gfCNCPoint1[15648] = {X 518.0643, Y 36.2972, Z -1.3333, A 0.000, B 0.000, C 0.000 }
gfCNCPoint1[15649] = {X 518.9098, Y 36.0014, Z -1.3333, A 0.000, B 0.000, C 0.000 }
gfCNCPoint1[15650] = {X 519.7999, Y 35.9011, Z -1.3333, A 0.000, B 0.000, C 0.000 }
gfCNCPoint1[15651] = {X 520.5225, Y 35.9015, Z -1.3333, A 0.000, B 0.000, C 0.000 }
gfCNCPoint1[15652] = {X 521.3209, Y 35.9930, Z -1.3333, A 0.000, B 0.000, C 0.000 }
gfCNCPoint1[15653] = {X 522.0848, Y 36.2423, Z -1.3333, A 0.000, B 0.000, C 0.000 }
gfCNCPoint1[15654] = {X 522.7835, Y 36.6393, Z -1.3333, A 0.000, B 0.000, C 0.000 }
gfCNCPoint1[15655] = {X 523.3887, Y 37.1679, Z -1.3333, A 0.000, B 0.000, C 0.000 }
gfCNCPoint1[15656] = {X 523.8761, Y 37.8068, Z -1.3333, A 0.000, B 0.000, C 0.000 }
gfCNCPoint1[15657] = {X 534.9519, Y 37.8074, Z -1.3333, A 0.000, B 0.000, C 0.000 }
gfCNCPoint1[15658] = {X 534.9519, Y 34.0445, Z -1.3333, A 0.000, B 0.000, C 0.000 }
gfCNCPoint1[15659] = {X 534.9533, Y 33.6446, Z -1.3333, A 0.000, B 0.000, C 0.000 }
gfCNCPoint1[15660] = {X 529.9327, Y 33.6439, Z -1.3333, A 0.000, B 0.000, C 0.000 }
gfCNCPoint1[15661] = {X 529.8235, Y 33.8172, Z -1.3333, A 0.000, B 0.000, C 0.000 }
gfCNCPoint1[15662] = {X 529.1840, Y 34.5408, Z -1.3333, A 0.000, B 0.000, C 0.000 }
gfCNCPoint1[15663] = {X 528.3897, Y 35.0900, Z -1.3333, A 0.000, B 0.000, C 0.000 }
gfCNCPoint1[15664] = {X 527.4869, Y 35.4329, Z -1.3333, A 0.000, B 0.000, C 0.000 }
gfCNCPoint1[15665] = {X 526.5282, Y 35.5495, Z -1.3333, A 0.000, B 0.000, C 0.000 }
gfCNCPoint1[15666] = {X 525.8868, Y 35.5495, Z -1.3333, A 0.000, B 0.000, C 0.000 }
gfCNCPoint1[15667] = {X 524.9967, Y 35.4492, Z -1.3333, A 0.000, B 0.000, C 0.000 }
gfCNCPoint1[15668] = {X 524.1512, Y 35.1533, Z -1.3333, A 0.000, B 0.000, C 0.000 }
gfCNCPoint1[15669] = {X 523.3928, Y 34.6768, Z -1.3333, A 0.000, B 0.000, C 0.000 }
gfCNCPoint1[15670] = {X 522.7594, Y 34.0434, Z -1.3333, A 0.000, B 0.000, C 0.000 }
gfCNCPoint1[15671] = {X 522.2829, Y 33.2850, Z -1.3333, A 0.000, B 0.000, C 0.000 }
gfCNCPoint1[15672] = {X 521.9870, Y 32.4395, Z -1.3333, A 0.000, B 0.000, C 0.000 }
gfCNCPoint1[15673] = {X 521.8868, Y 31.5495, Z -1.3333, A 0.000, B 0.000, C 0.000 }
gfCNCPoint1[15674] = {X 521.8868, Y 24.5714, Z -1.3333, A 0.000, B 0.000, C 0.000 }
gfCNCPoint1[15675] = {X 521.9870, Y 23.6813, Z -1.3333, A 0.000, B 0.000, C 0.000 }
gfCNCPoint1[15676] = {X 522.2829, Y 22.8359, Z -1.3333, A 0.000, B 0.000, C 0.000 }
gfCNCPoint1[15677] = {X 522.7594, Y 22.0775, Z -1.3333, A 0.000, B 0.000, C 0.000 }
gfCNCPoint1[15678] = {X 523.3928, Y 21.4441, Z -1.3333, A 0.000, B 0.000, C 0.000 }
gfCNCPoint1[15679] = {X 524.1512, Y 20.9675, Z -1.3333, A 0.000, B 0.000, C 0.000 }
gfCNCPoint1[15680] = {X 524.9967, Y 20.6717, Z -1.3333, A 0.000, B 0.000, C 0.000 }
gfCNCPoint1[15681] = {X 525.8868, Y 20.5714, Z -1.3333, A 0.000, B 0.000, C 0.000 }
gfCNCPoint1[15682] = {X 526.5664, Y 20.5716, Z -1.3333, A 0.000, B 0.000, C 0.000 }
gfCNCPoint1[15683] = {X 527.3632, Y 20.6595, Z -1.3333, A 0.000, B 0.000, C 0.000 }
gfCNCPoint1[15684] = {X 528.1265, Y 20.9045, Z -1.3333, A 0.000, B 0.000, C 0.000 }
gfCNCPoint1[15685] = {X 528.8256, Y 21.2968, Z -1.3333, A 0.000, B 0.000, C 0.000 }
gfCNCPoint1[15686] = {X 529.4324, Y 21.8207, Z -1.3333, A 0.000, B 0.000, C 0.000 }
gfCNCPoint1[15687] = {X 529.9226, Y 22.4550, Z -1.3333, A 0.000, B 0.000, C 0.000 }
gfCNCPoint1[15688] = {X 534.9519, Y 22.4554, Z -1.3333, A 0.000, B 0.000, C 0.000 }
gfCNCPoint1[15689] = {X 534.9519, Y 19.7809, Z -1.3333, A 0.000, B 0.000, C 0.000 }
gfCNCPoint1[15690] = {X 534.9534, Y 19.3810, Z -1.3333, A 0.000, B 0.000, C 0.000 }
gfCNCPoint1[15691] = {X 524.0161, Y 19.3804, Z -1.3333, A 0.000, B 0.000, C 0.000 }
gfCNCPoint1[15692] = {X 523.9057, Y 19.5536, Z -1.3333, A 0.000, B 0.000, C 0.000 }
gfCNCPoint1[15693] = {X 523.2662, Y 20.2771, Z -1.3333, A 0.000, B 0.000, C 0.000 }
gfCNCPoint1[15694] = {X 522.4720, Y 20.8263, Z -1.3333, A 0.000, B 0.000, C 0.000 }
gfCNCPoint1[15695] = {X 521.5693, Y 21.1692, Z -1.3333, A 0.000, B 0.000, C 0.000 }
gfCNCPoint1[15696] = {X 520.6107, Y 21.2857, Z -1.3333, A 0.000, B 0.000, C 0.000 }
gfCNCPoint1[15697] = {X 519.9691, Y 21.2857, Z -1.3333, A 0.000, B 0.000, C 0.000 }
gfCNCPoint1[15698] = {X 519.0790, Y 21.1854, Z -1.3333, A 0.000, B 0.000, C 0.000 }
gfCNCPoint1[15699] = {X 518.2336, Y 20.8896, Z -1.3333, A 0.000, B 0.000, C 0.000 }
gfCNCPoint1[15700] = {X 517.4751, Y 20.4130, Z -1.3333, A 0.000, B 0.000, C 0.000 }
gfCNCPoint1[15701] = {X 516.8418, Y 19.7797, Z -1.3333, A 0.000, B 0.000, C 0.000 }
gfCNCPoint1[15702] = {X 516.3652, Y 19.0212, Z -1.3333, A 0.000, B 0.000, C 0.000 }
gfCNCPoint1[15703] = {X 516.0694, Y 18.1758, Z -1.3333, A 0.000, B 0.000, C 0.000 }
gfCNCPoint1[15704] = {X 515.9691, Y 17.2857, Z -1.3333, A 0.000, B 0.000, C 0.000 }
gfCNCPoint1[15705] = {X 515.9691, Y 10.3077, Z -1.3333, A 0.000, B 0.000, C 0.000 }
gfCNCPoint1[15706] = {X 516.0694, Y 9.4176, Z -1.3333, A 0.000, B 0.000, C 0.000 }
gfCNCPoint1[15707] = {X 516.3652, Y 8.5721, Z -1.3333, A 0.000, B 0.000, C 0.000 }
gfCNCPoint1[15708] = {X 516.8418, Y 7.8137, Z -1.3333, A 0.000, B 0.000, C 0.000 }
gfCNCPoint1[15709] = {X 517.4752, Y 7.1803, Z -1.3333, A 0.000, B 0.000, C 0.000 }
gfCNCPoint1[15710] = {X 518.2337, Y 6.7038, Z -1.3333, A 0.000, B 0.000, C 0.000 }
gfCNCPoint1[15711] = {X 519.0791, Y 6.4080, Z -1.3333, A 0.000, B 0.000, C 0.000 }
gfCNCPoint1[15712] = {X 519.9693, Y 6.3077, Z -1.3333, A 0.000, B 0.000, C 0.000 }
gfCNCPoint1[15713] = {X 520.6473, Y 6.3079, Z -1.3333, A 0.000, B 0.000, C 0.000 }
gfCNCPoint1[15714] = {X 521.4444, Y 6.3955, Z -1.3333, A 0.000, B 0.000, C 0.000 }
gfCNCPoint1[15715] = {X 522.2081, Y 6.6404, Z -1.3333, A 0.000, B 0.000, C 0.000 }
gfCNCPoint1[15716] = {X 522.9075, Y 7.0328, Z -1.3333, A 0.000, B 0.000, C 0.000 }
gfCNCPoint1[15717] = {X 523.5146, Y 7.5567, Z -1.3333, A 0.000, B 0.000, C 0.000 }
gfCNCPoint1[15718] = {X 524.0050, Y 8.1913, Z -1.3333, A 0.000, B 0.000, C 0.000 }
gfCNCPoint1[15719] = {X 533.9641, Y 8.1916, Z -1.3333, A 0.000, B 0.000, C 0.000 }
gfCNCPoint1[15720] = {X 533.9642, Y 4.1116, Z -1.3333, A 0.000, B 0.000, C 0.000 }
gfCNCPoint1[15721] = {X 533.9642, Y 4.1116, Z 1.6667, A 0.000, B 0.000, C 0.000 }
gfCNCPoint1[15722] = {X 533.9642, Y 4.1116, Z 11.0000, A 0.000, B 0.000, C 0.000 }
gfCNCPoint1[15723] = {X 419.6130, Y 26.5284, Z 11.0000, A 0.000, B 0.000, C 0.000 }
gfCNCPoint1[15724] = {X 419.6130, Y 26.5284, Z 1.6667, A 0.000, B 0.000, C 0.000 }
gfCNCPoint1[15725] = {X 419.6130, Y 26.5284, Z -1.3333, A 0.000, B 0.000, C 0.000 }
gfCNCPoint1[15726] = {X 416.1497, Y 24.3716, Z -1.3333, A 0.000, B 0.000, C 0.000 }
gfCNCPoint1[15727] = {X 411.5457, Y 31.7648, Z -1.3333, A 0.000, B 0.000, C 0.000 }
gfCNCPoint1[15728] = {X 411.5464, Y 40.8985, Z -1.3333, A 0.000, B 0.000, C 0.000 }
gfCNCPoint1[15729] = {X 412.1845, Y 41.5843, Z -1.3333, A 0.000, B 0.000, C 0.000 }
gfCNCPoint1[15730] = {X 412.6648, Y 42.3885, Z -1.3333, A 0.000, B 0.000, C 0.000 }
gfCNCPoint1[15731] = {X 412.9660, Y 43.2755, Z -1.3333, A 0.000, B 0.000, C 0.000 }
gfCNCPoint1[15732] = {X 413.0747, Y 44.2059, Z -1.3333, A 0.000, B 0.000, C 0.000 }
gfCNCPoint1[15733] = {X 413.0747, Y 45.0002, Z -1.3333, A 0.000, B 0.000, C 0.000 }
gfCNCPoint1[15734] = {X 412.9663, Y 45.9614, Z -1.3333, A 0.000, B 0.000, C 0.000 }
gfCNCPoint1[15735] = {X 412.6468, Y 46.8745, Z -1.3333, A 0.000, B 0.000, C 0.000 }
gfCNCPoint1[15736] = {X 412.1321, Y 47.6935, Z -1.3333, A 0.000, B 0.000, C 0.000 }
gfCNCPoint1[15737] = {X 411.4481, Y 48.3776, Z -1.3333, A 0.000, B 0.000, C 0.000 }
gfCNCPoint1[15738] = {X 410.6290, Y 48.8922, Z -1.3333, A 0.000, B 0.000, C 0.000 }
gfCNCPoint1[15739] = {X 409.7159, Y 49.2117, Z -1.3333, A 0.000, B 0.000, C 0.000 }
gfCNCPoint1[15740] = {X 408.7547, Y 49.3200, Z -1.3333, A 0.000, B 0.000, C 0.000 }
gfCNCPoint1[15741] = {X 402.3112, Y 49.3200, Z -1.3333, A 0.000, B 0.000, C 0.000 }
gfCNCPoint1[15742] = {X 401.3546, Y 49.2127, Z -1.3333, A 0.000, B 0.000, C 0.000 }
gfCNCPoint1[15743] = {X 400.4455, Y 48.8963, Z -1.3333, A 0.000, B 0.000, C 0.000 }
gfCNCPoint1[15744] = {X 399.6290, Y 48.3864, Z -1.3333, A 0.000, B 0.000, C 0.000 }
gfCNCPoint1[15745] = {X 398.9457, Y 47.7084, Z -1.3333, A 0.000, B 0.000, C 0.000 }
gfCNCPoint1[15746] = {X 398.4295, Y 46.8959, Z -1.3333, A 0.000, B 0.000, C 0.000 }
gfCNCPoint1[15747] = {X 398.1060, Y 45.9892, Z -1.3333, A 0.000, B 0.000, C 0.000 }
gfCNCPoint1[15748] = {X 397.9913, Y 45.0335, Z -1.3333, A 0.000, B 0.000, C 0.000 }
gfCNCPoint1[15749] = {X 397.9916, Y 44.1528, Z -1.3333, A 0.000, B 0.000, C 0.000 }
gfCNCPoint1[15750] = {X 398.1015, Y 43.2391, Z -1.3333, A 0.000, B 0.000, C 0.000 }
gfCNCPoint1[15751] = {X 398.4024, Y 42.3694, Z -1.3333, A 0.000, B 0.000, C 0.000 }
gfCNCPoint1[15752] = {X 398.8807, Y 41.5832, Z -1.3333, A 0.000, B 0.000, C 0.000 }
gfCNCPoint1[15753] = {X 399.5147, Y 40.9161, Z -1.3333, A 0.000, B 0.000, C 0.000 }
gfCNCPoint1[15754] = {X 399.4729, Y 31.5978, Z -1.3333, A 0.000, B 0.000, C 0.000 }
gfCNCPoint1[15755] = {X 393.3550, Y 20.9593, Z -1.3333, A 0.000, B 0.000, C 0.000 }
gfCNCPoint1[15756] = {X 392.5218, Y 19.5476, Z -1.3333, A 0.000, B 0.000, C 0.000 }
gfCNCPoint1[15757] = {X 391.6571, Y 18.1549, Z -1.3333, A 0.000, B 0.000, C 0.000 }
gfCNCPoint1[15758] = {X 391.2004, Y 17.5289, Z -1.3333, A 0.000, B 0.000, C 0.000 }
gfCNCPoint1[15759] = {X 390.6680, Y 16.9657, Z -1.3333, A 0.000, B 0.000, C 0.000 }
gfCNCPoint1[15760] = {X 389.7910, Y 16.4734, Z -1.3333, A 0.000, B 0.000, C 0.000 }
gfCNCPoint1[15761] = {X 389.0515, Y 15.7916, Z -1.3333, A 0.000, B 0.000, C 0.000 }
gfCNCPoint1[15762] = {X 388.4898, Y 14.9574, Z -1.3333, A 0.000, B 0.000, C 0.000 }
gfCNCPoint1[15763] = {X 388.1361, Y 14.0158, Z -1.3333, A 0.000, B 0.000, C 0.000 }
gfCNCPoint1[15764] = {X 388.0098, Y 13.0180, Z -1.3333, A 0.000, B 0.000, C 0.000 }
gfCNCPoint1[15765] = {X 388.0096, Y 12.1868, Z -1.3333, A 0.000, B 0.000, C 0.000 }
gfCNCPoint1[15766] = {X 388.1179, Y 11.2255, Z -1.3333, A 0.000, B 0.000, C 0.000 }
gfCNCPoint1[15767] = {X 388.4374, Y 10.3125, Z -1.3333, A 0.000, B 0.000, C 0.000 }
gfCNCPoint1[15768] = {X 388.9521, Y 9.4933, Z -1.3333, A 0.000, B 0.000, C 0.000 }
gfCNCPoint1[15769] = {X 389.6361, Y 8.8093, Z -1.3333, A 0.000, B 0.000, C 0.000 }
gfCNCPoint1[15770] = {X 390.4552, Y 8.2946, Z -1.3333, A 0.000, B 0.000, C 0.000 }
gfCNCPoint1[15771] = {X 391.3683, Y 7.9751, Z -1.3333, A 0.000, B 0.000, C 0.000 }
gfCNCPoint1[15772] = {X 392.3296, Y 7.8668, Z -1.3333, A 0.000, B 0.000, C 0.000 }
gfCNCPoint1[15773] = {X 399.1118, Y 7.8668, Z -1.3333, A 0.000, B 0.000, C 0.000 }
gfCNCPoint1[15774] = {X 400.0730, Y 7.9751, Z -1.3333, A 0.000, B 0.000, C 0.000 }
gfCNCPoint1[15775] = {X 400.9861, Y 8.2946, Z -1.3333, A 0.000, B 0.000, C 0.000 }
gfCNCPoint1[15776] = {X 401.8052, Y 8.8093, Z -1.3333, A 0.000, B 0.000, C 0.000 }
gfCNCPoint1[15777] = {X 402.4893, Y 9.4933, Z -1.3333, A 0.000, B 0.000, C 0.000 }
gfCNCPoint1[15778] = {X 403.0039, Y 10.3124, Z -1.3333, A 0.000, B 0.000, C 0.000 }
gfCNCPoint1[15779] = {X 403.3234, Y 11.2255, Z -1.3333, A 0.000, B 0.000, C 0.000 }
gfCNCPoint1[15780] = {X 403.4318, Y 12.1868, Z -1.3333, A 0.000, B 0.000, C 0.000 }
gfCNCPoint1[15781] = {X 403.4318, Y 12.9781, Z -1.3333, A 0.000, B 0.000, C 0.000 }
gfCNCPoint1[15782] = {X 403.3293, Y 13.9134, Z -1.3333, A 0.000, B 0.000, C 0.000 }
gfCNCPoint1[15783] = {X 403.0267, Y 14.8043, Z -1.3333, A 0.000, B 0.000, C 0.000 }
gfCNCPoint1[15784] = {X 405.3573, Y 18.8239, Z -1.3333, A 0.000, B 0.000, C 0.000 }
gfCNCPoint1[15785] = {X 407.8738, Y 14.7547, Z -1.3333, A 0.000, B 0.000, C 0.000 }
gfCNCPoint1[15786] = {X 407.5921, Y 13.9048, Z -1.3333, A 0.000, B 0.000, C 0.000 }
gfCNCPoint1[15787] = {X 407.4917, Y 13.0151, Z -1.3333, A 0.000, B 0.000, C 0.000 }
gfCNCPoint1[15788] = {X 407.4915, Y 12.1868, Z -1.3333, A 0.000, B 0.000, C 0.000 }
gfCNCPoint1[15789] = {X 407.5999, Y 11.2255, Z -1.3333, A 0.000, B 0.000, C 0.000 }
gfCNCPoint1[15790] = {X 407.9194, Y 10.3124, Z -1.3333, A 0.000, B 0.000, C 0.000 }
gfCNCPoint1[15791] = {X 408.4340, Y 9.4933, Z -1.3333, A 0.000, B 0.000, C 0.000 }
gfCNCPoint1[15792] = {X 409.1181, Y 8.8093, Z -1.3333, A 0.000, B 0.000, C 0.000 }
gfCNCPoint1[15793] = {X 409.9372, Y 8.2946, Z -1.3333, A 0.000, B 0.000, C 0.000 }
gfCNCPoint1[15794] = {X 410.8502, Y 7.9751, Z -1.3333, A 0.000, B 0.000, C 0.000 }
gfCNCPoint1[15795] = {X 411.8115, Y 7.8668, Z -1.3333, A 0.000, B 0.000, C 0.000 }
gfCNCPoint1[15796] = {X 419.3245, Y 7.8668, Z -1.3333, A 0.000, B 0.000, C 0.000 }
gfCNCPoint1[15797] = {X 420.2858, Y 7.9751, Z -1.3333, A 0.000, B 0.000, C 0.000 }
gfCNCPoint1[15798] = {X 421.1988, Y 8.2946, Z -1.3333, A 0.000, B 0.000, C 0.000 }
gfCNCPoint1[15799] = {X 422.0179, Y 8.8093, Z -1.3333, A 0.000, B 0.000, C 0.000 }
gfCNCPoint1[15800] = {X 422.7020, Y 9.4933, Z -1.3333, A 0.000, B 0.000, C 0.000 }
gfCNCPoint1[15801] = {X 423.2166, Y 10.3124, Z -1.3333, A 0.000, B 0.000, C 0.000 }
gfCNCPoint1[15802] = {X 423.5361, Y 11.2255, Z -1.3333, A 0.000, B 0.000, C 0.000 }
gfCNCPoint1[15803] = {X 423.6445, Y 12.1868, Z -1.3333, A 0.000, B 0.000, C 0.000 }
gfCNCPoint1[15804] = {X 423.6444, Y 12.9805, Z -1.3333, A 0.000, B 0.000, C 0.000 }
gfCNCPoint1[15805] = {X 423.5509, Y 13.8470, Z -1.3333, A 0.000, B 0.000, C 0.000 }
gfCNCPoint1[15806] = {X 423.2879, Y 14.6778, Z -1.3333, A 0.000, B 0.000, C 0.000 }
gfCNCPoint1[15807] = {X 422.8659, Y 15.4403, Z -1.3333, A 0.000, B 0.000, C 0.000 }
gfCNCPoint1[15808] = {X 422.3016, Y 16.1044, Z -1.3333, A 0.000, B 0.000, C 0.000 }
gfCNCPoint1[15809] = {X 421.6172, Y 16.6439, Z -1.3333, A 0.000, B 0.000, C 0.000 }
gfCNCPoint1[15810] = {X 420.8396, Y 17.0375, Z -1.3333, A 0.000, B 0.000, C 0.000 }
gfCNCPoint1[15811] = {X 420.1233, Y 18.0010, Z -1.3333, A 0.000, B 0.000, C 0.000 }
gfCNCPoint1[15812] = {X 419.4749, Y 19.0115, Z -1.3333, A 0.000, B 0.000, C 0.000 }
gfCNCPoint1[15813] = {X 417.9942, Y 21.4097, Z -1.3333, A 0.000, B 0.000, C 0.000 }
gfCNCPoint1[15814] = {X 416.1497, Y 24.3716, Z -1.3333, A 0.000, B 0.000, C 0.000 }
gfCNCPoint1[15815] = {X 419.5451, Y 26.4861, Z -1.3333, A 0.000, B 0.000, C 0.000 }
gfCNCPoint1[15816] = {X 416.0818, Y 24.3293, Z -1.3333, A 0.000, B 0.000, C 0.000 }
gfCNCPoint1[15817] = {X 411.4657, Y 31.7419, Z -1.3333, A 0.000, B 0.000, C 0.000 }
gfCNCPoint1[15818] = {X 411.4664, Y 40.9352, Z -1.3333, A 0.000, B 0.000, C 0.000 }
gfCNCPoint1[15819] = {X 412.1041, Y 41.6106, Z -1.3333, A 0.000, B 0.000, C 0.000 }
gfCNCPoint1[15820] = {X 412.5845, Y 42.4056, Z -1.3333, A 0.000, B 0.000, C 0.000 }
gfCNCPoint1[15821] = {X 412.8859, Y 43.2842, Z -1.3333, A 0.000, B 0.000, C 0.000 }
gfCNCPoint1[15822] = {X 412.9947, Y 44.2068, Z -1.3333, A 0.000, B 0.000, C 0.000 }
gfCNCPoint1[15823] = {X 412.9947, Y 45.0001, Z -1.3333, A 0.000, B 0.000, C 0.000 }
gfCNCPoint1[15824] = {X 412.8883, Y 45.9436, Z -1.3333, A 0.000, B 0.000, C 0.000 }
gfCNCPoint1[15825] = {X 412.5747, Y 46.8398, Z -1.3333, A 0.000, B 0.000, C 0.000 }
gfCNCPoint1[15826] = {X 412.0696, Y 47.6437, Z -1.3333, A 0.000, B 0.000, C 0.000 }
gfCNCPoint1[15827] = {X 411.3982, Y 48.3150, Z -1.3333, A 0.000, B 0.000, C 0.000 }
gfCNCPoint1[15828] = {X 410.5943, Y 48.8201, Z -1.3333, A 0.000, B 0.000, C 0.000 }
gfCNCPoint1[15829] = {X 409.6981, Y 49.1337, Z -1.3333, A 0.000, B 0.000, C 0.000 }
gfCNCPoint1[15830] = {X 408.7547, Y 49.2400, Z -1.3333, A 0.000, B 0.000, C 0.000 }
gfCNCPoint1[15831] = {X 402.3112, Y 49.2400, Z -1.3333, A 0.000, B 0.000, C 0.000 }
gfCNCPoint1[15832] = {X 401.3723, Y 49.1347, Z -1.3333, A 0.000, B 0.000, C 0.000 }
gfCNCPoint1[15833] = {X 400.4800, Y 48.8242, Z -1.3333, A 0.000, B 0.000, C 0.000 }
gfCNCPoint1[15834] = {X 399.6786, Y 48.3237, Z -1.3333, A 0.000, B 0.000, C 0.000 }
gfCNCPoint1[15835] = {X 399.0080, Y 47.6582, Z -1.3333, A 0.000, B 0.000, C 0.000 }
gfCNCPoint1[15836] = {X 398.5013, Y 46.8608, Z -1.3333, A 0.000, B 0.000, C 0.000 }
gfCNCPoint1[15837] = {X 398.1839, Y 45.9709, Z -1.3333, A 0.000, B 0.000, C 0.000 }
gfCNCPoint1[15838] = {X 398.0713, Y 45.0329, Z -1.3333, A 0.000, B 0.000, C 0.000 }
gfCNCPoint1[15839] = {X 398.0716, Y 44.1538, Z -1.3333, A 0.000, B 0.000, C 0.000 }
gfCNCPoint1[15840] = {X 398.1815, Y 43.2480, Z -1.3333, A 0.000, B 0.000, C 0.000 }
gfCNCPoint1[15841] = {X 398.4827, Y 42.3867, Z -1.3333, A 0.000, B 0.000, C 0.000 }
gfCNCPoint1[15842] = {X 398.9612, Y 41.6098, Z -1.3333, A 0.000, B 0.000, C 0.000 }
gfCNCPoint1[15843] = {X 399.5948, Y 40.9532, Z -1.3333, A 0.000, B 0.000, C 0.000 }
gfCNCPoint1[15844] = {X 399.5528, Y 31.5762, Z -1.3333, A 0.000, B 0.000, C 0.000 }
gfCNCPoint1[15845] = {X 393.4243, Y 20.9194, Z -1.3333, A 0.000, B 0.000, C 0.000 }
gfCNCPoint1[15846] = {X 392.5903, Y 19.5061, Z -1.3333, A 0.000, B 0.000, C 0.000 }
gfCNCPoint1[15847] = {X 391.7246, Y 18.1119, Z -1.3333, A 0.000, B 0.000, C 0.000 }
gfCNCPoint1[15848] = {X 391.2572, Y 17.4721, Z -1.3333, A 0.000, B 0.000, C 0.000 }
gfCNCPoint1[15849] = {X 390.7119, Y 16.8973, Z -1.3333, A 0.000, B 0.000, C 0.000 }
gfCNCPoint1[15850] = {X 389.8472, Y 16.4153, Z -1.3333, A 0.000, B 0.000, C 0.000 }
gfCNCPoint1[15851] = {X 389.1178, Y 15.7460, Z -1.3333, A 0.000, B 0.000, C 0.000 }
gfCNCPoint1[15852] = {X 388.5635, Y 14.9258, Z -1.3333, A 0.000, B 0.000, C 0.000 }
gfCNCPoint1[15853] = {X 388.2145, Y 13.9994, Z -1.3333, A 0.000, B 0.000, C 0.000 }
gfCNCPoint1[15854] = {X 388.0898, Y 13.0173, Z -1.3333, A 0.000, B 0.000, C 0.000 }
gfCNCPoint1[15855] = {X 388.0896, Y 12.1868, Z -1.3333, A 0.000, B 0.000, C 0.000 }
gfCNCPoint1[15856] = {X 388.1959, Y 11.2433, Z -1.3333, A 0.000, B 0.000, C 0.000 }
gfCNCPoint1[15857] = {X 388.5095, Y 10.3472, Z -1.3333, A 0.000, B 0.000, C 0.000 }
gfCNCPoint1[15858] = {X 389.0147, Y 9.5432, Z -1.3333, A 0.000, B 0.000, C 0.000 }
gfCNCPoint1[15859] = {X 389.6860, Y 8.8719, Z -1.3333, A 0.000, B 0.000, C 0.000 }
gfCNCPoint1[15860] = {X 390.4900, Y 8.3667, Z -1.3333, A 0.000, B 0.000, C 0.000 }
gfCNCPoint1[15861] = {X 391.3861, Y 8.0531, Z -1.3333, A 0.000, B 0.000, C 0.000 }
gfCNCPoint1[15862] = {X 392.3296, Y 7.9468, Z -1.3333, A 0.000, B 0.000, C 0.000 }
gfCNCPoint1[15863] = {X 399.1118, Y 7.9468, Z -1.3333, A 0.000, B 0.000, C 0.000 }
gfCNCPoint1[15864] = {X 400.0552, Y 8.0531, Z -1.3333, A 0.000, B 0.000, C 0.000 }
gfCNCPoint1[15865] = {X 400.9514, Y 8.3667, Z -1.3333, A 0.000, B 0.000, C 0.000 }
gfCNCPoint1[15866] = {X 401.7554, Y 8.8718, Z -1.3333, A 0.000, B 0.000, C 0.000 }
gfCNCPoint1[15867] = {X 402.4267, Y 9.5432, Z -1.3333, A 0.000, B 0.000, C 0.000 }
gfCNCPoint1[15868] = {X 402.9319, Y 10.3471, Z -1.3333, A 0.000, B 0.000, C 0.000 }
gfCNCPoint1[15869] = {X 403.2455, Y 11.2433, Z -1.3333, A 0.000, B 0.000, C 0.000 }
gfCNCPoint1[15870] = {X 403.3518, Y 12.1868, Z -1.3333, A 0.000, B 0.000, C 0.000 }
gfCNCPoint1[15871] = {X 403.3518, Y 12.9781, Z -1.3333, A 0.000, B 0.000, C 0.000 }
gfCNCPoint1[15872] = {X 403.2466, Y 13.9164, Z -1.3333, A 0.000, B 0.000, C 0.000 }
gfCNCPoint1[15873] = {X 402.9365, Y 14.8081, Z -1.3333, A 0.000, B 0.000, C 0.000 }
gfCNCPoint1[15874] = {X 405.3551, Y 18.9796, Z -1.3333, A 0.000, B 0.000, C 0.000 }
gfCNCPoint1[15875] = {X 407.9643, Y 14.7603, Z -1.3333, A 0.000, B 0.000, C 0.000 }
gfCNCPoint1[15876] = {X 407.6749, Y 13.9083, Z -1.3333, A 0.000, B 0.000, C 0.000 }
gfCNCPoint1[15877] = {X 407.5717, Y 13.0144, Z -1.3333, A 0.000, B 0.000, C 0.000 }
gfCNCPoint1[15878] = {X 407.5715, Y 12.1868, Z -1.3333, A 0.000, B 0.000, C 0.000 }
gfCNCPoint1[15879] = {X 407.6778, Y 11.2433, Z -1.3333, A 0.000, B 0.000, C 0.000 }
gfCNCPoint1[15880] = {X 407.9914, Y 10.3471, Z -1.3333, A 0.000, B 0.000, C 0.000 }
gfCNCPoint1[15881] = {X 408.4966, Y 9.5432, Z -1.3333, A 0.000, B 0.000, C 0.000 }
gfCNCPoint1[15882] = {X 409.1679, Y 8.8718, Z -1.3333, A 0.000, B 0.000, C 0.000 }
gfCNCPoint1[15883] = {X 409.9719, Y 8.3667, Z -1.3333, A 0.000, B 0.000, C 0.000 }
gfCNCPoint1[15884] = {X 410.8680, Y 8.0531, Z -1.3333, A 0.000, B 0.000, C 0.000 }
gfCNCPoint1[15885] = {X 411.8115, Y 7.9468, Z -1.3333, A 0.000, B 0.000, C 0.000 }
gfCNCPoint1[15886] = {X 419.3245, Y 7.9468, Z -1.3333, A 0.000, B 0.000, C 0.000 }
gfCNCPoint1[15887] = {X 420.2679, Y 8.0531, Z -1.3333, A 0.000, B 0.000, C 0.000 }
gfCNCPoint1[15888] = {X 421.1641, Y 8.3667, Z -1.3333, A 0.000, B 0.000, C 0.000 }
gfCNCPoint1[15889] = {X 421.9681, Y 8.8718, Z -1.3333, A 0.000, B 0.000, C 0.000 }
gfCNCPoint1[15890] = {X 422.6394, Y 9.5432, Z -1.3333, A 0.000, B 0.000, C 0.000 }
gfCNCPoint1[15891] = {X 423.1446, Y 10.3471, Z -1.3333, A 0.000, B 0.000, C 0.000 }
gfCNCPoint1[15892] = {X 423.4582, Y 11.2433, Z -1.3333, A 0.000, B 0.000, C 0.000 }
gfCNCPoint1[15893] = {X 423.5645, Y 12.1868, Z -1.3333, A 0.000, B 0.000, C 0.000 }
gfCNCPoint1[15894] = {X 423.5645, Y 12.9799, Z -1.3333, A 0.000, B 0.000, C 0.000 }
gfCNCPoint1[15895] = {X 423.4718, Y 13.8340, Z -1.3333, A 0.000, B 0.000, C 0.000 }
gfCNCPoint1[15896] = {X 423.2116, Y 14.6528, Z -1.3333, A 0.000, B 0.000, C 0.000 }
gfCNCPoint1[15897] = {X 422.7940, Y 15.4037, Z -1.3333, A 0.000, B 0.000, C 0.000 }
gfCNCPoint1[15898] = {X 422.2357, Y 16.0568, Z -1.3333, A 0.000, B 0.000, C 0.000 }
gfCNCPoint1[15899] = {X 421.5590, Y 16.5861, Z -1.3333, A 0.000, B 0.000, C 0.000 }
gfCNCPoint1[15900] = {X 420.7907, Y 16.9706, Z -1.3333, A 0.000, B 0.000, C 0.000 }
gfCNCPoint1[15901] = {X 420.0639, Y 17.9463, Z -1.3333, A 0.000, B 0.000, C 0.000 }
gfCNCPoint1[15902] = {X 419.4065, Y 18.9701, Z -1.3333, A 0.000, B 0.000, C 0.000 }
gfCNCPoint1[15903] = {X 417.9262, Y 21.3675, Z -1.3333, A 0.000, B 0.000, C 0.000 }
gfCNCPoint1[15904] = {X 416.0818, Y 24.3293, Z -1.3333, A 0.000, B 0.000, C 0.000 }
gfCNCPoint1[15905] = {X 419.4772, Y 26.4438, Z -1.3333, A 0.000, B 0.000, C 0.000 }
gfCNCPoint1[15906] = {X 416.0139, Y 24.2870, Z -1.3333, A 0.000, B 0.000, C 0.000 }
gfCNCPoint1[15907] = {X 411.3857, Y 31.7190, Z -1.3333, A 0.000, B 0.000, C 0.000 }
gfCNCPoint1[15908] = {X 411.3864, Y 40.9722, Z -1.3333, A 0.000, B 0.000, C 0.000 }
gfCNCPoint1[15909] = {X 412.0237, Y 41.6371, Z -1.3333, A 0.000, B 0.000, C 0.000 }
gfCNCPoint1[15910] = {X 412.5042, Y 42.4228, Z -1.3333, A 0.000, B 0.000, C 0.000 }
gfCNCPoint1[15911] = {X 412.8059, Y 43.2931, Z -1.3333, A 0.000, B 0.000, C 0.000 }
gfCNCPoint1[15912] = {X 412.9147, Y 44.2076, Z -1.3333, A 0.000, B 0.000, C 0.000 }
gfCNCPoint1[15913] = {X 412.9147, Y 45.0001, Z -1.3333, A 0.000, B 0.000, C 0.000 }
gfCNCPoint1[15914] = {X 412.8104, Y 45.9258, Z -1.3333, A 0.000, B 0.000, C 0.000 }
gfCNCPoint1[15915] = {X 412.5027, Y 46.8051, Z -1.3333, A 0.000, B 0.000, C 0.000 }
gfCNCPoint1[15916] = {X 412.0070, Y 47.5938, Z -1.3333, A 0.000, B 0.000, C 0.000 }
gfCNCPoint1[15917] = {X 411.3483, Y 48.2525, Z -1.3333, A 0.000, B 0.000, C 0.000 }
gfCNCPoint1[15918] = {X 410.5596, Y 48.7480, Z -1.3333, A 0.000, B 0.000, C 0.000 }
gfCNCPoint1[15919] = {X 409.6803, Y 49.0557, Z -1.3333, A 0.000, B 0.000, C 0.000 }
gfCNCPoint1[15920] = {X 408.7547, Y 49.1600, Z -1.3333, A 0.000, B 0.000, C 0.000 }
gfCNCPoint1[15921] = {X 402.3112, Y 49.1600, Z -1.3333, A 0.000, B 0.000, C 0.000 }
gfCNCPoint1[15922] = {X 401.3900, Y 49.0567, Z -1.3333, A 0.000, B 0.000, C 0.000 }
gfCNCPoint1[15923] = {X 400.5146, Y 48.7520, Z -1.3333, A 0.000, B 0.000, C 0.000 }
gfCNCPoint1[15924] = {X 399.7283, Y 48.2610, Z -1.3333, A 0.000, B 0.000, C 0.000 }
gfCNCPoint1[15925] = {X 399.0703, Y 47.6081, Z -1.3333, A 0.000, B 0.000, C 0.000 }
gfCNCPoint1[15926] = {X 398.5732, Y 46.8257, Z -1.3333, A 0.000, B 0.000, C 0.000 }
gfCNCPoint1[15927] = {X 398.2617, Y 45.9526, Z -1.3333, A 0.000, B 0.000, C 0.000 }
gfCNCPoint1[15928] = {X 398.1513, Y 45.0322, Z -1.3333, A 0.000, B 0.000, C 0.000 }
gfCNCPoint1[15929] = {X 398.1516, Y 44.1549, Z -1.3333, A 0.000, B 0.000, C 0.000 }
gfCNCPoint1[15930] = {X 398.2616, Y 43.2570, Z -1.3333, A 0.000, B 0.000, C 0.000 }
gfCNCPoint1[15931] = {X 398.5630, Y 42.4041, Z -1.3333, A 0.000, B 0.000, C 0.000 }
gfCNCPoint1[15932] = {X 399.0417, Y 41.6366, Z -1.3333, A 0.000, B 0.000, C 0.000 }
gfCNCPoint1[15933] = {X 399.6750, Y 40.9907, Z -1.3333, A 0.000, B 0.000, C 0.000 }
gfCNCPoint1[15934] = {X 399.6327, Y 31.5547, Z -1.3333, A 0.000, B 0.000, C 0.000 }
gfCNCPoint1[15935] = {X 393.4937, Y 20.8796, Z -1.3333, A 0.000, B 0.000, C 0.000 }
gfCNCPoint1[15936] = {X 392.6587, Y 19.4647, Z -1.3333, A 0.000, B 0.000, C 0.000 }
gfCNCPoint1[15937] = {X 391.7921, Y 18.0690, Z -1.3333, A 0.000, B 0.000, C 0.000 }
gfCNCPoint1[15938] = {X 391.3140, Y 17.4153, Z -1.3333, A 0.000, B 0.000, C 0.000 }
gfCNCPoint1[15939] = {X 390.7557, Y 16.8288, Z -1.3333, A 0.000, B 0.000, C 0.000 }
gfCNCPoint1[15940] = {X 389.9033, Y 16.3572, Z -1.3333, A 0.000, B 0.000, C 0.000 }
gfCNCPoint1[15941] = {X 389.1840, Y 15.7003, Z -1.3333, A 0.000, B 0.000, C 0.000 }
gfCNCPoint1[15942] = {X 388.6372, Y 14.8941, Z -1.3333, A 0.000, B 0.000, C 0.000 }
gfCNCPoint1[15943] = {X 388.2928, Y 13.9829, Z -1.3333, A 0.000, B 0.000, C 0.000 }
gfCNCPoint1[15944] = {X 388.1698, Y 13.0166, Z -1.3333, A 0.000, B 0.000, C 0.000 }
gfCNCPoint1[15945] = {X 388.1696, Y 12.1868, Z -1.3333, A 0.000, B 0.000, C 0.000 }
gfCNCPoint1[15946] = {X 388.2739, Y 11.2611, Z -1.3333, A 0.000, B 0.000, C 0.000 }
gfCNCPoint1[15947] = {X 388.5816, Y 10.3819, Z -1.3333, A 0.000, B 0.000, C 0.000 }
gfCNCPoint1[15948] = {X 389.0772, Y 9.5931, Z -1.3333, A 0.000, B 0.000, C 0.000 }
gfCNCPoint1[15949] = {X 389.7359, Y 8.9344, Z -1.3333, A 0.000, B 0.000, C 0.000 }
gfCNCPoint1[15950] = {X 390.5247, Y 8.4388, Z -1.3333, A 0.000, B 0.000, C 0.000 }
gfCNCPoint1[15951] = {X 391.4039, Y 8.1311, Z -1.3333, A 0.000, B 0.000, C 0.000 }
gfCNCPoint1[15952] = {X 392.3296, Y 8.0268, Z -1.3333, A 0.000, B 0.000, C 0.000 }
gfCNCPoint1[15953] = {X 399.1118, Y 8.0268, Z -1.3333, A 0.000, B 0.000, C 0.000 }
gfCNCPoint1[15954] = {X 400.0374, Y 8.1311, Z -1.3333, A 0.000, B 0.000, C 0.000 }
gfCNCPoint1[15955] = {X 400.9167, Y 8.4388, Z -1.3333, A 0.000, B 0.000, C 0.000 }
gfCNCPoint1[15956] = {X 401.7055, Y 8.9344, Z -1.3333, A 0.000, B 0.000, C 0.000 }
gfCNCPoint1[15957] = {X 402.3642, Y 9.5931, Z -1.3333, A 0.000, B 0.000, C 0.000 }
gfCNCPoint1[15958] = {X 402.8598, Y 10.3819, Z -1.3333, A 0.000, B 0.000, C 0.000 }
gfCNCPoint1[15959] = {X 403.1675, Y 11.2611, Z -1.3333, A 0.000, B 0.000, C 0.000 }
gfCNCPoint1[15960] = {X 403.2718, Y 12.1868, Z -1.3333, A 0.000, B 0.000, C 0.000 }
gfCNCPoint1[15961] = {X 403.2718, Y 12.9781, Z -1.3333, A 0.000, B 0.000, C 0.000 }
gfCNCPoint1[15962] = {X 403.1639, Y 13.9192, Z -1.3333, A 0.000, B 0.000, C 0.000 }
gfCNCPoint1[15963] = {X 402.8459, Y 14.8115, Z -1.3333, A 0.000, B 0.000, C 0.000 }
gfCNCPoint1[15964] = {X 405.3529, Y 19.1352, Z -1.3333, A 0.000, B 0.000, C 0.000 }
gfCNCPoint1[15965] = {X 408.0552, Y 14.7656, Z -1.3333, A 0.000, B 0.000, C 0.000 }
gfCNCPoint1[15966] = {X 407.7577, Y 13.9117, Z -1.3333, A 0.000, B 0.000, C 0.000 }
gfCNCPoint1[15967] = {X 407.6517, Y 13.0137, Z -1.3333, A 0.000, B 0.000, C 0.000 }
gfCNCPoint1[15968] = {X 407.6515, Y 12.1868, Z -1.3333, A 0.000, B 0.000, C 0.000 }
gfCNCPoint1[15969] = {X 407.7558, Y 11.2611, Z -1.3333, A 0.000, B 0.000, C 0.000 }
gfCNCPoint1[15970] = {X 408.0635, Y 10.3819, Z -1.3333, A 0.000, B 0.000, C 0.000 }
gfCNCPoint1[15971] = {X 408.5591, Y 9.5931, Z -1.3333, A 0.000, B 0.000, C 0.000 }
gfCNCPoint1[15972] = {X 409.2178, Y 8.9344, Z -1.3333, A 0.000, B 0.000, C 0.000 }
gfCNCPoint1[15973] = {X 410.0066, Y 8.4388, Z -1.3333, A 0.000, B 0.000, C 0.000 }
gfCNCPoint1[15974] = {X 410.8859, Y 8.1311, Z -1.3333, A 0.000, B 0.000, C 0.000 }
gfCNCPoint1[15975] = {X 411.8115, Y 8.0268, Z -1.3333, A 0.000, B 0.000, C 0.000 }
gfCNCPoint1[15976] = {X 419.3245, Y 8.0268, Z -1.3333, A 0.000, B 0.000, C 0.000 }
gfCNCPoint1[15977] = {X 420.2501, Y 8.1311, Z -1.3333, A 0.000, B 0.000, C 0.000 }
gfCNCPoint1[15978] = {X 421.1294, Y 8.4388, Z -1.3333, A 0.000, B 0.000, C 0.000 }
gfCNCPoint1[15979] = {X 421.9182, Y 8.9344, Z -1.3333, A 0.000, B 0.000, C 0.000 }
gfCNCPoint1[15980] = {X 422.5769, Y 9.5931, Z -1.3333, A 0.000, B 0.000, C 0.000 }
gfCNCPoint1[15981] = {X 423.0725, Y 10.3819, Z -1.3333, A 0.000, B 0.000, C 0.000 }
gfCNCPoint1[15982] = {X 423.3802, Y 11.2611, Z -1.3333, A 0.000, B 0.000, C 0.000 }
gfCNCPoint1[15983] = {X 423.4845, Y 12.1868, Z -1.3333, A 0.000, B 0.000, C 0.000 }
gfCNCPoint1[15984] = {X 423.4845, Y 12.9792, Z -1.3333, A 0.000, B 0.000, C 0.000 }
gfCNCPoint1[15985] = {X 423.3928, Y 13.8211, Z -1.3333, A 0.000, B 0.000, C 0.000 }
gfCNCPoint1[15986] = {X 423.1352, Y 14.6277, Z -1.3333, A 0.000, B 0.000, C 0.000 }
gfCNCPoint1[15987] = {X 422.7221, Y 15.3669, Z -1.3333, A 0.000, B 0.000, C 0.000 }
gfCNCPoint1[15988] = {X 422.1700, Y 16.0090, Z -1.3333, A 0.000, B 0.000, C 0.000 }
gfCNCPoint1[15989] = {X 421.5010, Y 16.5281, Z -1.3333, A 0.000, B 0.000, C 0.000 }
gfCNCPoint1[15990] = {X 420.7419, Y 16.9035, Z -1.3333, A 0.000, B 0.000, C 0.000 }
gfCNCPoint1[15991] = {X 420.0046, Y 17.8915, Z -1.3333, A 0.000, B 0.000, C 0.000 }
gfCNCPoint1[15992] = {X 419.3380, Y 18.9286, Z -1.3333, A 0.000, B 0.000, C 0.000 }
gfCNCPoint1[15993] = {X 417.8583, Y 21.3253, Z -1.3333, A 0.000, B 0.000, C 0.000 }
gfCNCPoint1[15994] = {X 416.0139, Y 24.2870, Z -1.3333, A 0.000, B 0.000, C 0.000 }
gfCNCPoint1[15995] = {X 419.4093, Y 26.4015, Z -1.3333, A 0.000, B 0.000, C 0.000 }
gfCNCPoint1[15996] = {X 415.9460, Y 24.2448, Z -1.3333, A 0.000, B 0.000, C 0.000 }
gfCNCPoint1[15997] = {X 411.3057, Y 31.6961, Z -1.3333, A 0.000, B 0.000, C 0.000 }
gfCNCPoint1[15998] = {X 411.3064, Y 41.0097, Z -1.3333, A 0.000, B 0.000, C 0.000 }
gfCNCPoint1[15999] = {X 411.9432, Y 41.6640, Z -1.3333, A 0.000, B 0.000, C 0.000 }
gfCNCPoint1[16000] = {X 412.4239, Y 42.4402, Z -1.3333, A 0.000, B 0.000, C 0.000 }
gfCNCPoint1[16001] = {X 412.7258, Y 43.3019, Z -1.3333, A 0.000, B 0.000, C 0.000 }
gfCNCPoint1[16002] = {X 412.8347, Y 44.2085, Z -1.3333, A 0.000, B 0.000, C 0.000 }
gfCNCPoint1[16003] = {X 412.8347, Y 45.0001, Z -1.3333, A 0.000, B 0.000, C 0.000 }
gfCNCPoint1[16004] = {X 412.7324, Y 45.9080, Z -1.3333, A 0.000, B 0.000, C 0.000 }
gfCNCPoint1[16005] = {X 412.4306, Y 46.7703, Z -1.3333, A 0.000, B 0.000, C 0.000 }
gfCNCPoint1[16006] = {X 411.9445, Y 47.5439, Z -1.3333, A 0.000, B 0.000, C 0.000 }
gfCNCPoint1[16007] = {X 411.2985, Y 48.1899, Z -1.3333, A 0.000, B 0.000, C 0.000 }
gfCNCPoint1[16008] = {X 410.5249, Y 48.6760, Z -1.3333, A 0.000, B 0.000, C 0.000 }
gfCNCPoint1[16009] = {X 409.6625, Y 48.9777, Z -1.3333, A 0.000, B 0.000, C 0.000 }
gfCNCPoint1[16010] = {X 408.7547, Y 49.0800, Z -1.3333, A 0.000, B 0.000, C 0.000 }
gfCNCPoint1[16011] = {X 402.3112, Y 49.0800, Z -1.3333, A 0.000, B 0.000, C 0.000 }
gfCNCPoint1[16012] = {X 401.4077, Y 48.9787, Z -1.3333, A 0.000, B 0.000, C 0.000 }
gfCNCPoint1[16013] = {X 400.5491, Y 48.6799, Z -1.3333, A 0.000, B 0.000, C 0.000 }
gfCNCPoint1[16014] = {X 399.7780, Y 48.1983, Z -1.3333, A 0.000, B 0.000, C 0.000 }
gfCNCPoint1[16015] = {X 399.1326, Y 47.5579, Z -1.3333, A 0.000, B 0.000, C 0.000 }
gfCNCPoint1[16016] = {X 398.6451, Y 46.7906, Z -1.3333, A 0.000, B 0.000, C 0.000 }
gfCNCPoint1[16017] = {X 398.3396, Y 45.9343, Z -1.3333, A 0.000, B 0.000, C 0.000 }
gfCNCPoint1[16018] = {X 398.2313, Y 45.0316, Z -1.3333, A 0.000, B 0.000, C 0.000 }
gfCNCPoint1[16019] = {X 398.2316, Y 44.1559, Z -1.3333, A 0.000, B 0.000, C 0.000 }
gfCNCPoint1[16020] = {X 398.3416, Y 43.2661, Z -1.3333, A 0.000, B 0.000, C 0.000 }
gfCNCPoint1[16021] = {X 398.6434, Y 42.4218, Z -1.3333, A 0.000, B 0.000, C 0.000 }
gfCNCPoint1[16022] = {X 399.1223, Y 41.6638, Z -1.3333, A 0.000, B 0.000, C 0.000 }
gfCNCPoint1[16023] = {X 399.7552, Y 41.0287, Z -1.3333, A 0.000, B 0.000, C 0.000 }
gfCNCPoint1[16024] = {X 399.7126, Y 31.5332, Z -1.3333, A 0.000, B 0.000, C 0.000 }
gfCNCPoint1[16025] = {X 393.5630, Y 20.8397, Z -1.3333, A 0.000, B 0.000, C 0.000 }
gfCNCPoint1[16026] = {X 392.7271, Y 19.4233, Z -1.3333, A 0.000, B 0.000, C 0.000 }
gfCNCPoint1[16027] = {X 391.8596, Y 18.0260, Z -1.3333, A 0.000, B 0.000, C 0.000 }
gfCNCPoint1[16028] = {X 391.3707, Y 17.3584, Z -1.3333, A 0.000, B 0.000, C 0.000 }
gfCNCPoint1[16029] = {X 390.7992, Y 16.7601, Z -1.3333, A 0.000, B 0.000, C 0.000 }
gfCNCPoint1[16030] = {X 389.9593, Y 16.2989, Z -1.3333, A 0.000, B 0.000, C 0.000 }
gfCNCPoint1[16031] = {X 389.2501, Y 15.6544, Z -1.3333, A 0.000, B 0.000, C 0.000 }
gfCNCPoint1[16032] = {X 388.7108, Y 14.8623, Z -1.3333, A 0.000, B 0.000, C 0.000 }
gfCNCPoint1[16033] = {X 388.3711, Y 13.9663, Z -1.3333, A 0.000, B 0.000, C 0.000 }
gfCNCPoint1[16034] = {X 388.2498, Y 13.0158, Z -1.3333, A 0.000, B 0.000, C 0.000 }
gfCNCPoint1[16035] = {X 388.2496, Y 12.1868, Z -1.3333, A 0.000, B 0.000, C 0.000 }
gfCNCPoint1[16036] = {X 388.3519, Y 11.2789, Z -1.3333, A 0.000, B 0.000, C 0.000 }
gfCNCPoint1[16037] = {X 388.6537, Y 10.4166, Z -1.3333, A 0.000, B 0.000, C 0.000 }
gfCNCPoint1[16038] = {X 389.1398, Y 9.6430, Z -1.3333, A 0.000, B 0.000, C 0.000 }
gfCNCPoint1[16039] = {X 389.7858, Y 8.9969, Z -1.3333, A 0.000, B 0.000, C 0.000 }
gfCNCPoint1[16040] = {X 390.5594, Y 8.5109, Z -1.3333, A 0.000, B 0.000, C 0.000 }
gfCNCPoint1[16041] = {X 391.4217, Y 8.2091, Z -1.3333, A 0.000, B 0.000, C 0.000 }
gfCNCPoint1[16042] = {X 392.3296, Y 8.1068, Z -1.3333, A 0.000, B 0.000, C 0.000 }
gfCNCPoint1[16043] = {X 399.1118, Y 8.1068, Z -1.3333, A 0.000, B 0.000, C 0.000 }
gfCNCPoint1[16044] = {X 400.0196, Y 8.2091, Z -1.3333, A 0.000, B 0.000, C 0.000 }
gfCNCPoint1[16045] = {X 400.8820, Y 8.5109, Z -1.3333, A 0.000, B 0.000, C 0.000 }
gfCNCPoint1[16046] = {X 401.6556, Y 8.9969, Z -1.3333, A 0.000, B 0.000, C 0.000 }
gfCNCPoint1[16047] = {X 402.3016, Y 9.6430, Z -1.3333, A 0.000, B 0.000, C 0.000 }
gfCNCPoint1[16048] = {X 402.7877, Y 10.4166, Z -1.3333, A 0.000, B 0.000, C 0.000 }
gfCNCPoint1[16049] = {X 403.0895, Y 11.2789, Z -1.3333, A 0.000, B 0.000, C 0.000 }
gfCNCPoint1[16050] = {X 403.1918, Y 12.1868, Z -1.3333, A 0.000, B 0.000, C 0.000 }
gfCNCPoint1[16051] = {X 403.1918, Y 12.9781, Z -1.3333, A 0.000, B 0.000, C 0.000 }
gfCNCPoint1[16052] = {X 403.0811, Y 13.9218, Z -1.3333, A 0.000, B 0.000, C 0.000 }
gfCNCPoint1[16053] = {X 402.7551, Y 14.8144, Z -1.3333, A 0.000, B 0.000, C 0.000 }
gfCNCPoint1[16054] = {X 405.3507, Y 19.2909, Z -1.3333, A 0.000, B 0.000, C 0.000 }
gfCNCPoint1[16055] = {X 408.1463, Y 14.7703, Z -1.3333, A 0.000, B 0.000, C 0.000 }
gfCNCPoint1[16056] = {X 408.1096, Y 14.6934, Z -1.3333, A 0.000, B 0.000, C 0.000 }
gfCNCPoint1[16057] = {X 408.0746, Y 14.6156, Z -1.3333, A 0.000, B 0.000, C 0.000 }
gfCNCPoint1[16058] = {X 407.8219, Y 13.8317, Z -1.3333, A 0.000, B 0.000, C 0.000 }
gfCNCPoint1[16059] = {X 407.7317, Y 13.0131, Z -1.3333, A 0.000, B 0.000, C 0.000 }
gfCNCPoint1[16060] = {X 407.7315, Y 12.1868, Z -1.3333, A 0.000, B 0.000, C 0.000 }
gfCNCPoint1[16061] = {X 407.8338, Y 11.2789, Z -1.3333, A 0.000, B 0.000, C 0.000 }
gfCNCPoint1[16062] = {X 408.1356, Y 10.4166, Z -1.3333, A 0.000, B 0.000, C 0.000 }
gfCNCPoint1[16063] = {X 408.6217, Y 9.6430, Z -1.3333, A 0.000, B 0.000, C 0.000 }
gfCNCPoint1[16064] = {X 409.2677, Y 8.9969, Z -1.3333, A 0.000, B 0.000, C 0.000 }
gfCNCPoint1[16065] = {X 410.0413, Y 8.5109, Z -1.3333, A 0.000, B 0.000, C 0.000 }
gfCNCPoint1[16066] = {X 410.9037, Y 8.2091, Z -1.3333, A 0.000, B 0.000, C 0.000 }
gfCNCPoint1[16067] = {X 411.8115, Y 8.1068, Z -1.3333, A 0.000, B 0.000, C 0.000 }
gfCNCPoint1[16068] = {X 419.3245, Y 8.1068, Z -1.3333, A 0.000, B 0.000, C 0.000 }
gfCNCPoint1[16069] = {X 420.2323, Y 8.2091, Z -1.3333, A 0.000, B 0.000, C 0.000 }
gfCNCPoint1[16070] = {X 421.0947, Y 8.5109, Z -1.3333, A 0.000, B 0.000, C 0.000 }
gfCNCPoint1[16071] = {X 421.8683, Y 8.9969, Z -1.3333, A 0.000, B 0.000, C 0.000 }
gfCNCPoint1[16072] = {X 422.5143, Y 9.6430, Z -1.3333, A 0.000, B 0.000, C 0.000 }
gfCNCPoint1[16073] = {X 423.0004, Y 10.4166, Z -1.3333, A 0.000, B 0.000, C 0.000 }
gfCNCPoint1[16074] = {X 423.3022, Y 11.2789, Z -1.3333, A 0.000, B 0.000, C 0.000 }
gfCNCPoint1[16075] = {X 423.4045, Y 12.1868, Z -1.3333, A 0.000, B 0.000, C 0.000 }
gfCNCPoint1[16076] = {X 423.4045, Y 12.9786, Z -1.3333, A 0.000, B 0.000, C 0.000 }
gfCNCPoint1[16077] = {X 423.3138, Y 13.8080, Z -1.3333, A 0.000, B 0.000, C 0.000 }
gfCNCPoint1[16078] = {X 423.0589, Y 14.6026, Z -1.3333, A 0.000, B 0.000, C 0.000 }
gfCNCPoint1[16079] = {X 422.6503, Y 15.3300, Z -1.3333, A 0.000, B 0.000, C 0.000 }
gfCNCPoint1[16080] = {X 422.1043, Y 15.9610, Z -1.3333, A 0.000, B 0.000, C 0.000 }
gfCNCPoint1[16081] = {X 421.4431, Y 16.4699, Z -1.3333, A 0.000, B 0.000, C 0.000 }
gfCNCPoint1[16082] = {X 420.6934, Y 16.8362, Z -1.3333, A 0.000, B 0.000, C 0.000 }
gfCNCPoint1[16083] = {X 419.9453, Y 17.8366, Z -1.3333, A 0.000, B 0.000, C 0.000 }
gfCNCPoint1[16084] = {X 419.2696, Y 18.8872, Z -1.3333, A 0.000, B 0.000, C 0.000 }
gfCNCPoint1[16085] = {X 417.7903, Y 21.2832, Z -1.3333, A 0.000, B 0.000, C 0.000 }
gfCNCPoint1[16086] = {X 415.9460, Y 24.2448, Z -1.3333, A 0.000, B 0.000, C 0.000 }
gfCNCPoint1[16087] = {X 419.3414, Y 26.3592, Z -1.3333, A 0.000, B 0.000, C 0.000 }
gfCNCPoint1[16088] = {X 415.8781, Y 24.2025, Z -1.3333, A 0.000, B 0.000, C 0.000 }
gfCNCPoint1[16089] = {X 411.2257, Y 31.6733, Z -1.3333, A 0.000, B 0.000, C 0.000 }
gfCNCPoint1[16090] = {X 411.2264, Y 41.0476, Z -1.3333, A 0.000, B 0.000, C 0.000 }
gfCNCPoint1[16091] = {X 411.8627, Y 41.6910, Z -1.3333, A 0.000, B 0.000, C 0.000 }
gfCNCPoint1[16092] = {X 412.3435, Y 42.4576, Z -1.3333, A 0.000, B 0.000, C 0.000 }
gfCNCPoint1[16093] = {X 412.6457, Y 43.3106, Z -1.3333, A 0.000, B 0.000, C 0.000 }
gfCNCPoint1[16094] = {X 412.7547, Y 44.2089, Z -1.3333, A 0.000, B 0.000, C 0.000 }
gfCNCPoint1[16095] = {X 412.7545, Y 45.0384, Z -1.3333, A 0.000, B 0.000, C 0.000 }
gfCNCPoint1[16096] = {X 412.6469, Y 45.9222, Z -1.3333, A 0.000, B 0.000, C 0.000 }
gfCNCPoint1[16097] = {X 412.3466, Y 46.7602, Z -1.3333, A 0.000, B 0.000, C 0.000 }
gfCNCPoint1[16098] = {X 411.8683, Y 47.5111, Z -1.3333, A 0.000, B 0.000, C 0.000 }
gfCNCPoint1[16099] = {X 411.2357, Y 48.1376, Z -1.3333, A 0.000, B 0.000, C 0.000 }
gfCNCPoint1[16100] = {X 410.4803, Y 48.6086, Z -1.3333, A 0.000, B 0.000, C 0.000 }
gfCNCPoint1[16101] = {X 409.6394, Y 48.9009, Z -1.3333, A 0.000, B 0.000, C 0.000 }
gfCNCPoint1[16102] = {X 408.7547, Y 49.0000, Z -1.3333, A 0.000, B 0.000, C 0.000 }
gfCNCPoint1[16103] = {X 402.3112, Y 49.0000, Z -1.3333, A 0.000, B 0.000, C 0.000 }
gfCNCPoint1[16104] = {X 401.4211, Y 48.8997, Z -1.3333, A 0.000, B 0.000, C 0.000 }
gfCNCPoint1[16105] = {X 400.5757, Y 48.6039, Z -1.3333, A 0.000, B 0.000, C 0.000 }
gfCNCPoint1[16106] = {X 399.8172, Y 48.1273, Z -1.3333, A 0.000, B 0.000, C 0.000 }
gfCNCPoint1[16107] = {X 399.1839, Y 47.4939, Z -1.3333, A 0.000, B 0.000, C 0.000 }
gfCNCPoint1[16108] = {X 398.7073, Y 46.7355, Z -1.3333, A 0.000, B 0.000, C 0.000 }
gfCNCPoint1[16109] = {X 398.4115, Y 45.8900, Z -1.3333, A 0.000, B 0.000, C 0.000 }
gfCNCPoint1[16110] = {X 398.3112, Y 44.9999, Z -1.3333, A 0.000, B 0.000, C 0.000 }
gfCNCPoint1[16111] = {X 398.3115, Y 44.1569, Z -1.3333, A 0.000, B 0.000, C 0.000 }
gfCNCPoint1[16112] = {X 398.4217, Y 43.2753, Z -1.3333, A 0.000, B 0.000, C 0.000 }
gfCNCPoint1[16113] = {X 398.7237, Y 42.4397, Z -1.3333, A 0.000, B 0.000, C 0.000 }
gfCNCPoint1[16114] = {X 399.2028, Y 41.6913, Z -1.3333, A 0.000, B 0.000, C 0.000 }
gfCNCPoint1[16115] = {X 399.8352, Y 41.0672, Z -1.3333, A 0.000, B 0.000, C 0.000 }
gfCNCPoint1[16116] = {X 399.8352, Y 31.6238, Z -1.3333, A 0.000, B 0.000, C 0.000 }
gfCNCPoint1[16117] = {X 399.8386, Y 31.5919, Z -1.3333, A 0.000, B 0.000, C 0.000 }
gfCNCPoint1[16118] = {X 393.6324, Y 20.7998, Z -1.3333, A 0.000, B 0.000, C 0.000 }
gfCNCPoint1[16119] = {X 392.7956, Y 19.3818, Z -1.3333, A 0.000, B 0.000, C 0.000 }
gfCNCPoint1[16120] = {X 391.9271, Y 17.9831, Z -1.3333, A 0.000, B 0.000, C 0.000 }
gfCNCPoint1[16121] = {X 391.4274, Y 17.3015, Z -1.3333, A 0.000, B 0.000, C 0.000 }
gfCNCPoint1[16122] = {X 390.8426, Y 16.6913, Z -1.3333, A 0.000, B 0.000, C 0.000 }
gfCNCPoint1[16123] = {X 390.0091, Y 16.2361, Z -1.3333, A 0.000, B 0.000, C 0.000 }
gfCNCPoint1[16124] = {X 389.3064, Y 15.5972, Z -1.3333, A 0.000, B 0.000, C 0.000 }
gfCNCPoint1[16125] = {X 388.7742, Y 14.8107, Z -1.3333, A 0.000, B 0.000, C 0.000 }
gfCNCPoint1[16126] = {X 388.4423, Y 13.9209, Z -1.3333, A 0.000, B 0.000, C 0.000 }
gfCNCPoint1[16127] = {X 388.3296, Y 12.9779, Z -1.3333, A 0.000, B 0.000, C 0.000 }
gfCNCPoint1[16128] = {X 388.3296, Y 12.1868, Z -1.3333, A 0.000, B 0.000, C 0.000 }
gfCNCPoint1[16129] = {X 388.4299, Y 11.2967, Z -1.3333, A 0.000, B 0.000, C 0.000 }
gfCNCPoint1[16130] = {X 388.7258, Y 10.4513, Z -1.3333, A 0.000, B 0.000, C 0.000 }
gfCNCPoint1[16131] = {X 389.2023, Y 9.6929, Z -1.3333, A 0.000, B 0.000, C 0.000 }
gfCNCPoint1[16132] = {X 389.8357, Y 9.0595, Z -1.3333, A 0.000, B 0.000, C 0.000 }
gfCNCPoint1[16133] = {X 390.5941, Y 8.5829, Z -1.3333, A 0.000, B 0.000, C 0.000 }
gfCNCPoint1[16134] = {X 391.4395, Y 8.2871, Z -1.3333, A 0.000, B 0.000, C 0.000 }
gfCNCPoint1[16135] = {X 392.3296, Y 8.1868, Z -1.3333, A 0.000, B 0.000, C 0.000 }
gfCNCPoint1[16136] = {X 399.1118, Y 8.1868, Z -1.3333, A 0.000, B 0.000, C 0.000 }
gfCNCPoint1[16137] = {X 400.0018, Y 8.2871, Z -1.3333, A 0.000, B 0.000, C 0.000 }
gfCNCPoint1[16138] = {X 400.8473, Y 8.5829, Z -1.3333, A 0.000, B 0.000, C 0.000 }
gfCNCPoint1[16139] = {X 401.6057, Y 9.0595, Z -1.3333, A 0.000, B 0.000, C 0.000 }
gfCNCPoint1[16140] = {X 402.2391, Y 9.6929, Z -1.3333, A 0.000, B 0.000, C 0.000 }
gfCNCPoint1[16141] = {X 402.7156, Y 10.4513, Z -1.3333, A 0.000, B 0.000, C 0.000 }
gfCNCPoint1[16142] = {X 403.0115, Y 11.2967, Z -1.3333, A 0.000, B 0.000, C 0.000 }
gfCNCPoint1[16143] = {X 403.1118, Y 12.1868, Z -1.3333, A 0.000, B 0.000, C 0.000 }
gfCNCPoint1[16144] = {X 403.1115, Y 13.0192, Z -1.3333, A 0.000, B 0.000, C 0.000 }
gfCNCPoint1[16145] = {X 402.9933, Y 13.9442, Z -1.3333, A 0.000, B 0.000, C 0.000 }
gfCNCPoint1[16146] = {X 402.6641, Y 14.8167, Z -1.3333, A 0.000, B 0.000, C 0.000 }
gfCNCPoint1[16147] = {X 405.2576, Y 19.3199, Z -1.3333, A 0.000, B 0.000, C 0.000 }
gfCNCPoint1[16148] = {X 405.3720, Y 19.4087, Z -1.3333, A 0.000, B 0.000, C 0.000 }
gfCNCPoint1[16149] = {X 408.1959, Y 14.8343, Z -1.3333, A 0.000, B 0.000, C 0.000 }
gfCNCPoint1[16150] = {X 408.2428, Y 14.7847, Z -1.3333, A 0.000, B 0.000, C 0.000 }
gfCNCPoint1[16151] = {X 408.1939, Y 14.6848, Z -1.3333, A 0.000, B 0.000, C 0.000 }
gfCNCPoint1[16152] = {X 408.1479, Y 14.5835, Z -1.3333, A 0.000, B 0.000, C 0.000 }
gfCNCPoint1[16153] = {X 407.8965, Y 13.7982, Z -1.3333, A 0.000, B 0.000, C 0.000 }
gfCNCPoint1[16154] = {X 407.8115, Y 12.9779, Z -1.3333, A 0.000, B 0.000, C 0.000 }
gfCNCPoint1[16155] = {X 407.8115, Y 12.1868, Z -1.3333, A 0.000, B 0.000, C 0.000 }
gfCNCPoint1[16156] = {X 407.9118, Y 11.2967, Z -1.3333, A 0.000, B 0.000, C 0.000 }
gfCNCPoint1[16157] = {X 408.2077, Y 10.4513, Z -1.3333, A 0.000, B 0.000, C 0.000 }
gfCNCPoint1[16158] = {X 408.6842, Y 9.6929, Z -1.3333, A 0.000, B 0.000, C 0.000 }
gfCNCPoint1[16159] = {X 409.3176, Y 9.0595, Z -1.3333, A 0.000, B 0.000, C 0.000 }
gfCNCPoint1[16160] = {X 410.0760, Y 8.5829, Z -1.3333, A 0.000, B 0.000, C 0.000 }
gfCNCPoint1[16161] = {X 410.9215, Y 8.2871, Z -1.3333, A 0.000, B 0.000, C 0.000 }
gfCNCPoint1[16162] = {X 411.8115, Y 8.1868, Z -1.3333, A 0.000, B 0.000, C 0.000 }
gfCNCPoint1[16163] = {X 419.3245, Y 8.1868, Z -1.3333, A 0.000, B 0.000, C 0.000 }
gfCNCPoint1[16164] = {X 420.2145, Y 8.2871, Z -1.3333, A 0.000, B 0.000, C 0.000 }
gfCNCPoint1[16165] = {X 421.0600, Y 8.5829, Z -1.3333, A 0.000, B 0.000, C 0.000 }
gfCNCPoint1[16166] = {X 421.8184, Y 9.0595, Z -1.3333, A 0.000, B 0.000, C 0.000 }
gfCNCPoint1[16167] = {X 422.4518, Y 9.6929, Z -1.3333, A 0.000, B 0.000, C 0.000 }
gfCNCPoint1[16168] = {X 422.9283, Y 10.4513, Z -1.3333, A 0.000, B 0.000, C 0.000 }
gfCNCPoint1[16169] = {X 423.2242, Y 11.2967, Z -1.3333, A 0.000, B 0.000, C 0.000 }
gfCNCPoint1[16170] = {X 423.3245, Y 12.1868, Z -1.3333, A 0.000, B 0.000, C 0.000 }
gfCNCPoint1[16171] = {X 423.3245, Y 12.9779, Z -1.3333, A 0.000, B 0.000, C 0.000 }
gfCNCPoint1[16172] = {X 423.1971, Y 13.9553, Z -1.3333, A 0.000, B 0.000, C 0.000 }
gfCNCPoint1[16173] = {X 422.8385, Y 14.8733, Z -1.3333, A 0.000, B 0.000, C 0.000 }
gfCNCPoint1[16174] = {X 422.2696, Y 15.6782, Z -1.3333, A 0.000, B 0.000, C 0.000 }
gfCNCPoint1[16175] = {X 421.5238, Y 16.3226, Z -1.3333, A 0.000, B 0.000, C 0.000 }
gfCNCPoint1[16176] = {X 420.6450, Y 16.7687, Z -1.3333, A 0.000, B 0.000, C 0.000 }
gfCNCPoint1[16177] = {X 419.8861, Y 17.7815, Z -1.3333, A 0.000, B 0.000, C 0.000 }
gfCNCPoint1[16178] = {X 419.2012, Y 18.8457, Z -1.3333, A 0.000, B 0.000, C 0.000 }
gfCNCPoint1[16179] = {X 417.7223, Y 21.2410, Z -1.3333, A 0.000, B 0.000, C 0.000 }
gfCNCPoint1[16180] = {X 415.8781, Y 24.2025, Z -1.3333, A 0.000, B 0.000, C 0.000 }
gfCNCPoint1[16181] = {X 419.3414, Y 26.3592, Z -1.3333, A 0.000, B 0.000, C 0.000 }
gfCNCPoint1[16182] = {X 419.3414, Y 26.3592, Z 1.6667, A 0.000, B 0.000, C 0.000 }
gfCNCPoint1[16183] = {X 419.3414, Y 26.3592, Z 11.0000, A 0.000, B 0.000, C 0.000 }
gfCNCPoint1[16184] = {X 352.3257, Y -3.5333, Z 11.0000, A 0.000, B 0.000, C 0.000 }
gfCNCPoint1[16185] = {X 352.3257, Y -3.5333, Z 1.6667, A 0.000, B 0.000, C 0.000 }
gfCNCPoint1[16186] = {X 352.3257, Y -3.5333, Z -1.3333, A 0.000, B 0.000, C 0.000 }
gfCNCPoint1[16187] = {X 351.5854, Y 0.4790, Z -1.3333, A 0.000, B 0.000, C 0.000 }
gfCNCPoint1[16188] = {X 351.8684, Y 0.5312, Z -1.3333, A 0.000, B 0.000, C 0.000 }
gfCNCPoint1[16189] = {X 353.8028, Y 1.0173, Z -1.3333, A 0.000, B 0.000, C 0.000 }
gfCNCPoint1[16190] = {X 355.6825, Y 1.6844, Z -1.3333, A 0.000, B 0.000, C 0.000 }
gfCNCPoint1[16191] = {X 357.4905, Y 2.5266, Z -1.3333, A 0.000, B 0.000, C 0.000 }
gfCNCPoint1[16192] = {X 359.2106, Y 3.5363, Z -1.3333, A 0.000, B 0.000, C 0.000 }
gfCNCPoint1[16193] = {X 360.8273, Y 4.7044, Z -1.3333, A 0.000, B 0.000, C 0.000 }
gfCNCPoint1[16194] = {X 362.3261, Y 6.0205, Z -1.3333, A 0.000, B 0.000, C 0.000 }
gfCNCPoint1[16195] = {X 363.6935, Y 7.4726, Z -1.3333, A 0.000, B 0.000, C 0.000 }
gfCNCPoint1[16196] = {X 365.1633, Y 9.3695, Z -1.3333, A 0.000, B 0.000, C 0.000 }
gfCNCPoint1[16197] = {X 366.4424, Y 11.3999, Z -1.3333, A 0.000, B 0.000, C 0.000 }
gfCNCPoint1[16198] = {X 367.5185, Y 13.5449, Z -1.3333, A 0.000, B 0.000, C 0.000 }
gfCNCPoint1[16199] = {X 368.3816, Y 15.7840, Z -1.3333, A 0.000, B 0.000, C 0.000 }
gfCNCPoint1[16200] = {X 369.0235, Y 18.0963, Z -1.3333, A 0.000, B 0.000, C 0.000 }
gfCNCPoint1[16201] = {X 369.5021, Y 20.7273, Z -1.3333, A 0.000, B 0.000, C 0.000 }
gfCNCPoint1[16202] = {X 369.7569, Y 23.3894, Z -1.3333, A 0.000, B 0.000, C 0.000 }
gfCNCPoint1[16203] = {X 369.7859, Y 26.0634, Z -1.3333, A 0.000, B 0.000, C 0.000 }
gfCNCPoint1[16204] = {X 369.5891, Y 28.7303, Z -1.3333, A 0.000, B 0.000, C 0.000 }
gfCNCPoint1[16205] = {X 369.1677, Y 31.3711, Z -1.3333, A 0.000, B 0.000, C 0.000 }
gfCNCPoint1[16206] = {X 368.6439, Y 33.4757, Z -1.3333, A 0.000, B 0.000, C 0.000 }
gfCNCPoint1[16207] = {X 367.9361, Y 35.5258, Z -1.3333, A 0.000, B 0.000, C 0.000 }
gfCNCPoint1[16208] = {X 367.0498, Y 37.5052, Z -1.3333, A 0.000, B 0.000, C 0.000 }
gfCNCPoint1[16209] = {X 365.9921, Y 39.3986, Z -1.3333, A 0.000, B 0.000, C 0.000 }
gfCNCPoint1[16210] = {X 364.7711, Y 41.1911, Z -1.3333, A 0.000, B 0.000, C 0.000 }
gfCNCPoint1[16211] = {X 363.5441, Y 42.7032, Z -1.3333, A 0.000, B 0.000, C 0.000 }
gfCNCPoint1[16212] = {X 362.1893, Y 44.1018, Z -1.3333, A 0.000, B 0.000, C 0.000 }
gfCNCPoint1[16213] = {X 360.7169, Y 45.3762, Z -1.3333, A 0.000, B 0.000, C 0.000 }
gfCNCPoint1[16214] = {X 359.1385, Y 46.5165, Z -1.3333, A 0.000, B 0.000, C 0.000 }
gfCNCPoint1[16215] = {X 357.4661, Y 47.5140, Z -1.3333, A 0.000, B 0.000, C 0.000 }
gfCNCPoint1[16216] = {X 355.5055, Y 48.4043, Z -1.3333, A 0.000, B 0.000, C 0.000 }
gfCNCPoint1[16217] = {X 353.4693, Y 49.1042, Z -1.3333, A 0.000, B 0.000, C 0.000 }
gfCNCPoint1[16218] = {X 351.3757, Y 49.6074, Z -1.3333, A 0.000, B 0.000, C 0.000 }
gfCNCPoint1[16219] = {X 349.2438, Y 49.9095, Z -1.3333, A 0.000, B 0.000, C 0.000 }
gfCNCPoint1[16220] = {X 347.0929, Y 50.0076, Z -1.3333, A 0.000, B 0.000, C 0.000 }
gfCNCPoint1[16221] = {X 345.0263, Y 49.9727, Z -1.3333, A 0.000, B 0.000, C 0.000 }
gfCNCPoint1[16222] = {X 342.9706, Y 49.7588, Z -1.3333, A 0.000, B 0.000, C 0.000 }
gfCNCPoint1[16223] = {X 340.9411, Y 49.3673, Z -1.3333, A 0.000, B 0.000, C 0.000 }
gfCNCPoint1[16224] = {X 338.9533, Y 48.8013, Z -1.3333, A 0.000, B 0.000, C 0.000 }
gfCNCPoint1[16225] = {X 337.0220, Y 48.0650, Z -1.3333, A 0.000, B 0.000, C 0.000 }
gfCNCPoint1[16226] = {X 335.1619, Y 47.1639, Z -1.3333, A 0.000, B 0.000, C 0.000 }
gfCNCPoint1[16227] = {X 333.5790, Y 46.1853, Z -1.3333, A 0.000, B 0.000, C 0.000 }
gfCNCPoint1[16228] = {X 332.0763, Y 45.0874, Z -1.3333, A 0.000, B 0.000, C 0.000 }
gfCNCPoint1[16229] = {X 330.6627, Y 43.8769, Z -1.3333, A 0.000, B 0.000, C 0.000 }
gfCNCPoint1[16230] = {X 329.7216, Y 43.8765, Z -1.3333, A 0.000, B 0.000, C 0.000 }
gfCNCPoint1[16231] = {X 328.8028, Y 43.6722, Z -1.3333, A 0.000, B 0.000, C 0.000 }
gfCNCPoint1[16232] = {X 327.9502, Y 43.2738, Z -1.3333, A 0.000, B 0.000, C 0.000 }
gfCNCPoint1[16233] = {X 327.2040, Y 42.7002, Z -1.3333, A 0.000, B 0.000, C 0.000 }
gfCNCPoint1[16234] = {X 326.5808, Y 42.0925, Z -1.3333, A 0.000, B 0.000, C 0.000 }
gfCNCPoint1[16235] = {X 325.9523, Y 41.3190, Z -1.3333, A 0.000, B 0.000, C 0.000 }
gfCNCPoint1[16236] = {X 325.5179, Y 40.4220, Z -1.3333, A 0.000, B 0.000, C 0.000 }
gfCNCPoint1[16237] = {X 325.3006, Y 39.4493, Z -1.3333, A 0.000, B 0.000, C 0.000 }
gfCNCPoint1[16238] = {X 325.3120, Y 38.4527, Z -1.3333, A 0.000, B 0.000, C 0.000 }
gfCNCPoint1[16239] = {X 325.5514, Y 37.4852, Z -1.3333, A 0.000, B 0.000, C 0.000 }
gfCNCPoint1[16240] = {X 326.0062, Y 36.5984, Z -1.3333, A 0.000, B 0.000, C 0.000 }
gfCNCPoint1[16241] = {X 330.2648, Y 30.2313, Z -1.3333, A 0.000, B 0.000, C 0.000 }
gfCNCPoint1[16242] = {X 330.8696, Y 29.5246, Z -1.3333, A 0.000, B 0.000, C 0.000 }
gfCNCPoint1[16243] = {X 331.6116, Y 28.9637, Z -1.3333, A 0.000, B 0.000, C 0.000 }
gfCNCPoint1[16244] = {X 332.4564, Y 28.5747, Z -1.3333, A 0.000, B 0.000, C 0.000 }
gfCNCPoint1[16245] = {X 333.3649, Y 28.3755, Z -1.3333, A 0.000, B 0.000, C 0.000 }
gfCNCPoint1[16246] = {X 334.2951, Y 28.3754, Z -1.3333, A 0.000, B 0.000, C 0.000 }
gfCNCPoint1[16247] = {X 335.2036, Y 28.5744, Z -1.3333, A 0.000, B 0.000, C 0.000 }
gfCNCPoint1[16248] = {X 336.0486, Y 28.9633, Z -1.3333, A 0.000, B 0.000, C 0.000 }
gfCNCPoint1[16249] = {X 336.7907, Y 29.5240, Z -1.3333, A 0.000, B 0.000, C 0.000 }
gfCNCPoint1[16250] = {X 337.4284, Y 30.1382, Z -1.3333, A 0.000, B 0.000, C 0.000 }
gfCNCPoint1[16251] = {X 337.9530, Y 30.7613, Z -1.3333, A 0.000, B 0.000, C 0.000 }
gfCNCPoint1[16252] = {X 338.3513, Y 31.4717, Z -1.3333, A 0.000, B 0.000, C 0.000 }
gfCNCPoint1[16253] = {X 338.6092, Y 32.2443, Z -1.3333, A 0.000, B 0.000, C 0.000 }
gfCNCPoint1[16254] = {X 338.7175, Y 33.0516, Z -1.3333, A 0.000, B 0.000, C 0.000 }
gfCNCPoint1[16255] = {X 338.6724, Y 33.8649, Z -1.3333, A 0.000, B 0.000, C 0.000 }
gfCNCPoint1[16256] = {X 339.4352, Y 34.5565, Z -1.3333, A 0.000, B 0.000, C 0.000 }
gfCNCPoint1[16257] = {X 340.2325, Y 35.2081, Z -1.3333, A 0.000, B 0.000, C 0.000 }
gfCNCPoint1[16258] = {X 341.5298, Y 36.0604, Z -1.3333, A 0.000, B 0.000, C 0.000 }
gfCNCPoint1[16259] = {X 342.9375, Y 36.7144, Z -1.3333, A 0.000, B 0.000, C 0.000 }
gfCNCPoint1[16260] = {X 344.4256, Y 37.1561, Z -1.3333, A 0.000, B 0.000, C 0.000 }
gfCNCPoint1[16261] = {X 345.9621, Y 37.3761, Z -1.3333, A 0.000, B 0.000, C 0.000 }
gfCNCPoint1[16262] = {X 347.5143, Y 37.3696, Z -1.3333, A 0.000, B 0.000, C 0.000 }
gfCNCPoint1[16263] = {X 348.9587, Y 37.1759, Z -1.3333, A 0.000, B 0.000, C 0.000 }
gfCNCPoint1[16264] = {X 350.3520, Y 36.7490, Z -1.3333, A 0.000, B 0.000, C 0.000 }
gfCNCPoint1[16265] = {X 351.6570, Y 36.1003, Z -1.3333, A 0.000, B 0.000, C 0.000 }
gfCNCPoint1[16266] = {X 352.8385, Y 35.2473, Z -1.3333, A 0.000, B 0.000, C 0.000 }
gfCNCPoint1[16267] = {X 353.9892, Y 34.1268, Z -1.3333, A 0.000, B 0.000, C 0.000 }
gfCNCPoint1[16268] = {X 354.9851, Y 32.8667, Z -1.3333, A 0.000, B 0.000, C 0.000 }
gfCNCPoint1[16269] = {X 355.8095, Y 31.4883, Z -1.3333, A 0.000, B 0.000, C 0.000 }
gfCNCPoint1[16270] = {X 356.4486, Y 30.0148, Z -1.3333, A 0.000, B 0.000, C 0.000 }
gfCNCPoint1[16271] = {X 356.8915, Y 28.4709, Z -1.3333, A 0.000, B 0.000, C 0.000 }
gfCNCPoint1[16272] = {X 357.1648, Y 26.7827, Z -1.3333, A 0.000, B 0.000, C 0.000 }
gfCNCPoint1[16273] = {X 357.2761, Y 25.0762, Z -1.3333, A 0.000, B 0.000, C 0.000 }
gfCNCPoint1[16274] = {X 357.2244, Y 23.3668, Z -1.3333, A 0.000, B 0.000, C 0.000 }
gfCNCPoint1[16275] = {X 357.0102, Y 21.6701, Z -1.3333, A 0.000, B 0.000, C 0.000 }
gfCNCPoint1[16276] = {X 356.6739, Y 20.2206, Z -1.3333, A 0.000, B 0.000, C 0.000 }
gfCNCPoint1[16277] = {X 356.1608, Y 18.8238, Z -1.3333, A 0.000, B 0.000, C 0.000 }
gfCNCPoint1[16278] = {X 355.4789, Y 17.5012, Z -1.3333, A 0.000, B 0.000, C 0.000 }
gfCNCPoint1[16279] = {X 354.6385, Y 16.2732, Z -1.3333, A 0.000, B 0.000, C 0.000 }
gfCNCPoint1[16280] = {X 353.7525, Y 15.2850, Z -1.3333, A 0.000, B 0.000, C 0.000 }
gfCNCPoint1[16281] = {X 352.7341, Y 14.4339, Z -1.3333, A 0.000, B 0.000, C 0.000 }
gfCNCPoint1[16282] = {X 351.6043, Y 13.7375, Z -1.3333, A 0.000, B 0.000, C 0.000 }
gfCNCPoint1[16283] = {X 350.3863, Y 13.2101, Z -1.3333, A 0.000, B 0.000, C 0.000 }
gfCNCPoint1[16284] = {X 349.1054, Y 12.8627, Z -1.3333, A 0.000, B 0.000, C 0.000 }
gfCNCPoint1[16285] = {X 347.3449, Y 12.6438, Z -1.3333, A 0.000, B 0.000, C 0.000 }
gfCNCPoint1[16286] = {X 345.5709, Y 12.6598, Z -1.3333, A 0.000, B 0.000, C 0.000 }
gfCNCPoint1[16287] = {X 343.8145, Y 12.9102, Z -1.3333, A 0.000, B 0.000, C 0.000 }
gfCNCPoint1[16288] = {X 342.1068, Y 13.3908, Z -1.3333, A 0.000, B 0.000, C 0.000 }
gfCNCPoint1[16289] = {X 340.4775, Y 14.0929, Z -1.3333, A 0.000, B 0.000, C 0.000 }
gfCNCPoint1[16290] = {X 338.9555, Y 15.0044, Z -1.3333, A 0.000, B 0.000, C 0.000 }
gfCNCPoint1[16291] = {X 338.9169, Y 15.8492, Z -1.3333, A 0.000, B 0.000, C 0.000 }
gfCNCPoint1[16292] = {X 338.7145, Y 16.6703, Z -1.3333, A 0.000, B 0.000, C 0.000 }
gfCNCPoint1[16293] = {X 338.3561, Y 17.4362, Z -1.3333, A 0.000, B 0.000, C 0.000 }
gfCNCPoint1[16294] = {X 337.8552, Y 18.1176, Z -1.3333, A 0.000, B 0.000, C 0.000 }
gfCNCPoint1[16295] = {X 337.2313, Y 18.6884, Z -1.3333, A 0.000, B 0.000, C 0.000 }
gfCNCPoint1[16296] = {X 336.5140, Y 19.2162, Z -1.3333, A 0.000, B 0.000, C 0.000 }
gfCNCPoint1[16297] = {X 335.6982, Y 19.6754, Z -1.3333, A 0.000, B 0.000, C 0.000 }
gfCNCPoint1[16298] = {X 334.8027, Y 19.9480, Z -1.3333, A 0.000, B 0.000, C 0.000 }
gfCNCPoint1[16299] = {X 333.8694, Y 20.0213, Z -1.3333, A 0.000, B 0.000, C 0.000 }
gfCNCPoint1[16300] = {X 332.9422, Y 19.8919, Z -1.3333, A 0.000, B 0.000, C 0.000 }
gfCNCPoint1[16301] = {X 332.0647, Y 19.5657, Z -1.3333, A 0.000, B 0.000, C 0.000 }
gfCNCPoint1[16302] = {X 331.2781, Y 19.0582, Z -1.3333, A 0.000, B 0.000, C 0.000 }
gfCNCPoint1[16303] = {X 330.6193, Y 18.3931, Z -1.3333, A 0.000, B 0.000, C 0.000 }
gfCNCPoint1[16304] = {X 330.1192, Y 17.6017, Z -1.3333, A 0.000, B 0.000, C 0.000 }
gfCNCPoint1[16305] = {X 326.5942, Y 10.3502, Z -1.3333, A 0.000, B 0.000, C 0.000 }
gfCNCPoint1[16306] = {X 326.2930, Y 9.5271, Z -1.3333, A 0.000, B 0.000, C 0.000 }
gfCNCPoint1[16307] = {X 326.1640, Y 8.6602, Z -1.3333, A 0.000, B 0.000, C 0.000 }
gfCNCPoint1[16308] = {X 326.2128, Y 7.7851, Z -1.3333, A 0.000, B 0.000, C 0.000 }
gfCNCPoint1[16309] = {X 326.4371, Y 6.9378, Z -1.3333, A 0.000, B 0.000, C 0.000 }
gfCNCPoint1[16310] = {X 326.8279, Y 6.1532, Z -1.3333, A 0.000, B 0.000, C 0.000 }
gfCNCPoint1[16311] = {X 327.3690, Y 5.4637, Z -1.3333, A 0.000, B 0.000, C 0.000 }
gfCNCPoint1[16312] = {X 328.0381, Y 4.8976, Z -1.3333, A 0.000, B 0.000, C 0.000 }
gfCNCPoint1[16313] = {X 328.7084, Y 4.4385, Z -1.3333, A 0.000, B 0.000, C 0.000 }
gfCNCPoint1[16314] = {X 329.5890, Y 3.9827, Z -1.3333, A 0.000, B 0.000, C 0.000 }
gfCNCPoint1[16315] = {X 330.5504, Y 3.7397, Z -1.3333, A 0.000, B 0.000, C 0.000 }
gfCNCPoint1[16316] = {X 331.5419, Y 3.7222, Z -1.3333, A 0.000, B 0.000, C 0.000 }
gfCNCPoint1[16317] = {X 332.5112, Y 3.9314, Z -1.3333, A 0.000, B 0.000, C 0.000 }
gfCNCPoint1[16318] = {X 333.9978, Y 3.1018, Z -1.3333, A 0.000, B 0.000, C 0.000 }
gfCNCPoint1[16319] = {X 335.5315, Y 2.3629, Z -1.3333, A 0.000, B 0.000, C 0.000 }
gfCNCPoint1[16320] = {X 337.6677, Y 1.4964, Z -1.3333, A 0.000, B 0.000, C 0.000 }
gfCNCPoint1[16321] = {X 339.8715, Y 0.8203, Z -1.3333, A 0.000, B 0.000, C 0.000 }
gfCNCPoint1[16322] = {X 342.1262, Y 0.3400, Z -1.3333, A 0.000, B 0.000, C 0.000 }
gfCNCPoint1[16323] = {X 344.4142, Y 0.0591, Z -1.3333, A 0.000, B 0.000, C 0.000 }
gfCNCPoint1[16324] = {X 346.7181, Y -0.0202, Z -1.3333, A 0.000, B 0.000, C 0.000 }
gfCNCPoint1[16325] = {X 349.0200, Y 0.1026, Z -1.3333, A 0.000, B 0.000, C 0.000 }
gfCNCPoint1[16326] = {X 351.3024, Y 0.4268, Z -1.3333, A 0.000, B 0.000, C 0.000 }
gfCNCPoint1[16327] = {X 351.5854, Y 0.4790, Z -1.3333, A 0.000, B 0.000, C 0.000 }
gfCNCPoint1[16328] = {X 352.3112, Y -3.4546, Z -1.3333, A 0.000, B 0.000, C 0.000 }
gfCNCPoint1[16329] = {X 351.5709, Y 0.5577, Z -1.3333, A 0.000, B 0.000, C 0.000 }
gfCNCPoint1[16330] = {X 351.8532, Y 0.6098, Z -1.3333, A 0.000, B 0.000, C 0.000 }
gfCNCPoint1[16331] = {X 353.7802, Y 1.0940, Z -1.3333, A 0.000, B 0.000, C 0.000 }
gfCNCPoint1[16332] = {X 355.6526, Y 1.7586, Z -1.3333, A 0.000, B 0.000, C 0.000 }
gfCNCPoint1[16333] = {X 357.4537, Y 2.5976, Z -1.3333, A 0.000, B 0.000, C 0.000 }
gfCNCPoint1[16334] = {X 359.1671, Y 3.6034, Z -1.3333, A 0.000, B 0.000, C 0.000 }
gfCNCPoint1[16335] = {X 360.7776, Y 4.7671, Z -1.3333, A 0.000, B 0.000, C 0.000 }
gfCNCPoint1[16336] = {X 362.2706, Y 6.0781, Z -1.3333, A 0.000, B 0.000, C 0.000 }
gfCNCPoint1[16337] = {X 363.6327, Y 7.5246, Z -1.3333, A 0.000, B 0.000, C 0.000 }
gfCNCPoint1[16338] = {X 365.0978, Y 9.4153, Z -1.3333, A 0.000, B 0.000, C 0.000 }
gfCNCPoint1[16339] = {X 366.3727, Y 11.4392, Z -1.3333, A 0.000, B 0.000, C 0.000 }
gfCNCPoint1[16340] = {X 367.4453, Y 13.5772, Z -1.3333, A 0.000, B 0.000, C 0.000 }
gfCNCPoint1[16341] = {X 368.3056, Y 15.8091, Z -1.3333, A 0.000, B 0.000, C 0.000 }
gfCNCPoint1[16342] = {X 368.9454, Y 18.1139, Z -1.3333, A 0.000, B 0.000, C 0.000 }
gfCNCPoint1[16343] = {X 369.4229, Y 20.7383, Z -1.3333, A 0.000, B 0.000, C 0.000 }
gfCNCPoint1[16344] = {X 369.6770, Y 23.3936, Z -1.3333, A 0.000, B 0.000, C 0.000 }
gfCNCPoint1[16345] = {X 369.7060, Y 26.0609, Z -1.3333, A 0.000, B 0.000, C 0.000 }
gfCNCPoint1[16346] = {X 369.5096, Y 28.7211, Z -1.3333, A 0.000, B 0.000, C 0.000 }
gfCNCPoint1[16347] = {X 369.0893, Y 31.3552, Z -1.3333, A 0.000, B 0.000, C 0.000 }
gfCNCPoint1[16348] = {X 368.5672, Y 33.4529, Z -1.3333, A 0.000, B 0.000, C 0.000 }
gfCNCPoint1[16349] = {X 367.8617, Y 35.4963, Z -1.3333, A 0.000, B 0.000, C 0.000 }
gfCNCPoint1[16350] = {X 366.9783, Y 37.4694, Z -1.3333, A 0.000, B 0.000, C 0.000 }
gfCNCPoint1[16351] = {X 365.9240, Y 39.3566, Z -1.3333, A 0.000, B 0.000, C 0.000 }
gfCNCPoint1[16352] = {X 364.7070, Y 41.1433, Z -1.3333, A 0.000, B 0.000, C 0.000 }
gfCNCPoint1[16353] = {X 363.4845, Y 42.6498, Z -1.3333, A 0.000, B 0.000, C 0.000 }
gfCNCPoint1[16354] = {X 362.1346, Y 44.0433, Z -1.3333, A 0.000, B 0.000, C 0.000 }
gfCNCPoint1[16355] = {X 360.6677, Y 45.3131, Z -1.3333, A 0.000, B 0.000, C 0.000 }
gfCNCPoint1[16356] = {X 359.0951, Y 46.4493, Z -1.3333, A 0.000, B 0.000, C 0.000 }
gfCNCPoint1[16357] = {X 357.4288, Y 47.4432, Z -1.3333, A 0.000, B 0.000, C 0.000 }
gfCNCPoint1[16358] = {X 355.4751, Y 48.3302, Z -1.3333, A 0.000, B 0.000, C 0.000 }
gfCNCPoint1[16359] = {X 353.4460, Y 49.0276, Z -1.3333, A 0.000, B 0.000, C 0.000 }
gfCNCPoint1[16360] = {X 351.3598, Y 49.5290, Z -1.3333, A 0.000, B 0.000, C 0.000 }
gfCNCPoint1[16361] = {X 349.2353, Y 49.8299, Z -1.3333, A 0.000, B 0.000, C 0.000 }
gfCNCPoint1[16362] = {X 347.0919, Y 49.9276, Z -1.3333, A 0.000, B 0.000, C 0.000 }
gfCNCPoint1[16363] = {X 345.0322, Y 49.8929, Z -1.3333, A 0.000, B 0.000, C 0.000 }
gfCNCPoint1[16364] = {X 342.9833, Y 49.6798, Z -1.3333, A 0.000, B 0.000, C 0.000 }
gfCNCPoint1[16365] = {X 340.9606, Y 49.2897, Z -1.3333, A 0.000, B 0.000, C 0.000 }
gfCNCPoint1[16366] = {X 338.9794, Y 48.7256, Z -1.3333, A 0.000, B 0.000, C 0.000 }
gfCNCPoint1[16367] = {X 337.0545, Y 47.9919, Z -1.3333, A 0.000, B 0.000, C 0.000 }
gfCNCPoint1[16368] = {X 335.2006, Y 47.0939, Z -1.3333, A 0.000, B 0.000, C 0.000 }
gfCNCPoint1[16369] = {X 333.6131, Y 46.1118, Z -1.3333, A 0.000, B 0.000, C 0.000 }
gfCNCPoint1[16370] = {X 332.1065, Y 45.0094, Z -1.3333, A 0.000, B 0.000, C 0.000 }
gfCNCPoint1[16371] = {X 330.6902, Y 43.7933, Z -1.3333, A 0.000, B 0.000, C 0.000 }
gfCNCPoint1[16372] = {X 329.7574, Y 43.7999, Z -1.3333, A 0.000, B 0.000, C 0.000 }
gfCNCPoint1[16373] = {X 328.8458, Y 43.6023, Z -1.3333, A 0.000, B 0.000, C 0.000 }
gfCNCPoint1[16374] = {X 327.9995, Y 43.2102, Z -1.3333, A 0.000, B 0.000, C 0.000 }
gfCNCPoint1[16375] = {X 327.2594, Y 42.6425, Z -1.3333, A 0.000, B 0.000, C 0.000 }
gfCNCPoint1[16376] = {X 326.6366, Y 42.0352, Z -1.3333, A 0.000, B 0.000, C 0.000 }
gfCNCPoint1[16377] = {X 326.0198, Y 41.2760, Z -1.3333, A 0.000, B 0.000, C 0.000 }
gfCNCPoint1[16378] = {X 325.5934, Y 40.3956, Z -1.3333, A 0.000, B 0.000, C 0.000 }
gfCNCPoint1[16379] = {X 325.3802, Y 39.4410, Z -1.3333, A 0.000, B 0.000, C 0.000 }
gfCNCPoint1[16380] = {X 325.3913, Y 38.4628, Z -1.3333, A 0.000, B 0.000, C 0.000 }
gfCNCPoint1[16381] = {X 325.6264, Y 37.5133, Z -1.3333, A 0.000, B 0.000, C 0.000 }
gfCNCPoint1[16382] = {X 326.0727, Y 36.6429, Z -1.3333, A 0.000, B 0.000, C 0.000 }
gfCNCPoint1[16383] = {X 330.3309, Y 30.2764, Z -1.3333, A 0.000, B 0.000, C 0.000 }
gfCNCPoint1[16384] = {X 330.9244, Y 29.5828, Z -1.3333, A 0.000, B 0.000, C 0.000 }
gfCNCPoint1[16385] = {X 331.6527, Y 29.0324, Z -1.3333, A 0.000, B 0.000, C 0.000 }
gfCNCPoint1[16386] = {X 332.4819, Y 28.6505, Z -1.3333, A 0.000, B 0.000, C 0.000 }
gfCNCPoint1[16387] = {X 333.3736, Y 28.4550, Z -1.3333, A 0.000, B 0.000, C 0.000 }
gfCNCPoint1[16388] = {X 334.2865, Y 28.4549, Z -1.3333, A 0.000, B 0.000, C 0.000 }
gfCNCPoint1[16389] = {X 335.1782, Y 28.6502, Z -1.3333, A 0.000, B 0.000, C 0.000 }
gfCNCPoint1[16390] = {X 336.0075, Y 29.0319, Z -1.3333, A 0.000, B 0.000, C 0.000 }
gfCNCPoint1[16391] = {X 336.7358, Y 29.5823, Z -1.3333, A 0.000, B 0.000, C 0.000 }
gfCNCPoint1[16392] = {X 337.3723, Y 30.1953, Z -1.3333, A 0.000, B 0.000, C 0.000 }
gfCNCPoint1[16393] = {X 337.8919, Y 30.8136, Z -1.3333, A 0.000, B 0.000, C 0.000 }
gfCNCPoint1[16394] = {X 338.2849, Y 31.5193, Z -1.3333, A 0.000, B 0.000, C 0.000 }
gfCNCPoint1[16395] = {X 338.5368, Y 32.2866, Z -1.3333, A 0.000, B 0.000, C 0.000 }
gfCNCPoint1[16396] = {X 338.6388, Y 33.0878, Z -1.3333, A 0.000, B 0.000, C 0.000 }
gfCNCPoint1[16397] = {X 338.5869, Y 33.8938, Z -1.3333, A 0.000, B 0.000, C 0.000 }
gfCNCPoint1[16398] = {X 339.3672, Y 34.6035, Z -1.3333, A 0.000, B 0.000, C 0.000 }
gfCNCPoint1[16399] = {X 340.1836, Y 35.2714, Z -1.3333, A 0.000, B 0.000, C 0.000 }
gfCNCPoint1[16400] = {X 341.4905, Y 36.1301, Z -1.3333, A 0.000, B 0.000, C 0.000 }
gfCNCPoint1[16401] = {X 342.9087, Y 36.7890, Z -1.3333, A 0.000, B 0.000, C 0.000 }
gfCNCPoint1[16402] = {X 344.4078, Y 37.2341, Z -1.3333, A 0.000, B 0.000, C 0.000 }
gfCNCPoint1[16403] = {X 345.9557, Y 37.4559, Z -1.3333, A 0.000, B 0.000, C 0.000 }
gfCNCPoint1[16404] = {X 347.5195, Y 37.4495, Z -1.3333, A 0.000, B 0.000, C 0.000 }
gfCNCPoint1[16405] = {X 348.6880, Y 37.3121, Z -1.3333, A 0.000, B 0.000, C 0.000 }
gfCNCPoint1[16406] = {X 349.8285, Y 37.0230, Z -1.3333, A 0.000, B 0.000, C 0.000 }
gfCNCPoint1[16407] = {X 350.9214, Y 36.5873, Z -1.3333, A 0.000, B 0.000, C 0.000 }
gfCNCPoint1[16408] = {X 351.9480, Y 36.0124, Z -1.3333, A 0.000, B 0.000, C 0.000 }
gfCNCPoint1[16409] = {X 352.8905, Y 35.3082, Z -1.3333, A 0.000, B 0.000, C 0.000 }
gfCNCPoint1[16410] = {X 354.0486, Y 34.1803, Z -1.3333, A 0.000, B 0.000, C 0.000 }
gfCNCPoint1[16411] = {X 355.0510, Y 32.9120, Z -1.3333, A 0.000, B 0.000, C 0.000 }
gfCNCPoint1[16412] = {X 355.8807, Y 31.5247, Z -1.3333, A 0.000, B 0.000, C 0.000 }
gfCNCPoint1[16413] = {X 356.5239, Y 30.0416, Z -1.3333, A 0.000, B 0.000, C 0.000 }
gfCNCPoint1[16414] = {X 356.9697, Y 28.4877, Z -1.3333, A 0.000, B 0.000, C 0.000 }
gfCNCPoint1[16415] = {X 357.2442, Y 26.7920, Z -1.3333, A 0.000, B 0.000, C 0.000 }
gfCNCPoint1[16416] = {X 357.3561, Y 25.0777, Z -1.3333, A 0.000, B 0.000, C 0.000 }
gfCNCPoint1[16417] = {X 357.3042, Y 23.3607, Z -1.3333, A 0.000, B 0.000, C 0.000 }
gfCNCPoint1[16418] = {X 357.0890, Y 21.6563, Z -1.3333, A 0.000, B 0.000, C 0.000 }
gfCNCPoint1[16419] = {X 356.7504, Y 20.1973, Z -1.3333, A 0.000, B 0.000, C 0.000 }
gfCNCPoint1[16420] = {X 356.2340, Y 18.7913, Z -1.3333, A 0.000, B 0.000, C 0.000 }
gfCNCPoint1[16421] = {X 355.5475, Y 17.4601, Z -1.3333, A 0.000, B 0.000, C 0.000 }
gfCNCPoint1[16422] = {X 354.7016, Y 16.2240, Z -1.3333, A 0.000, B 0.000, C 0.000 }
gfCNCPoint1[16423] = {X 353.8080, Y 15.2273, Z -1.3333, A 0.000, B 0.000, C 0.000 }
gfCNCPoint1[16424] = {X 352.7807, Y 14.3689, Z -1.3333, A 0.000, B 0.000, C 0.000 }
gfCNCPoint1[16425] = {X 351.6411, Y 13.6665, Z -1.3333, A 0.000, B 0.000, C 0.000 }
gfCNCPoint1[16426] = {X 350.4126, Y 13.1346, Z -1.3333, A 0.000, B 0.000, C 0.000 }
gfCNCPoint1[16427] = {X 349.1206, Y 12.7841, Z -1.3333, A 0.000, B 0.000, C 0.000 }
gfCNCPoint1[16428] = {X 347.3420, Y 12.5636, Z -1.3333, A 0.000, B 0.000, C 0.000 }
gfCNCPoint1[16429] = {X 345.5499, Y 12.5812, Z -1.3333, A 0.000, B 0.000, C 0.000 }
gfCNCPoint1[16430] = {X 343.7759, Y 12.8366, Z -1.3333, A 0.000, B 0.000, C 0.000 }
gfCNCPoint1[16431] = {X 342.0517, Y 13.3254, Z -1.3333, A 0.000, B 0.000, C 0.000 }
gfCNCPoint1[16432] = {X 340.4076, Y 14.0389, Z -1.3333, A 0.000, B 0.000, C 0.000 }
gfCNCPoint1[16433] = {X 338.8728, Y 14.9645, Z -1.3333, A 0.000, B 0.000, C 0.000 }
gfCNCPoint1[16434] = {X 338.8756, Y 15.0086, Z -1.3333, A 0.000, B 0.000, C 0.000 }
gfCNCPoint1[16435] = {X 338.8378, Y 15.8377, Z -1.3333, A 0.000, B 0.000, C 0.000 }
gfCNCPoint1[16436] = {X 338.6391, Y 16.6436, Z -1.3333, A 0.000, B 0.000, C 0.000 }
gfCNCPoint1[16437] = {X 338.2873, Y 17.3954, Z -1.3333, A 0.000, B 0.000, C 0.000 }
gfCNCPoint1[16438] = {X 337.7957, Y 18.0642, Z -1.3333, A 0.000, B 0.000, C 0.000 }
gfCNCPoint1[16439] = {X 337.1833, Y 18.6244, Z -1.3333, A 0.000, B 0.000, C 0.000 }
gfCNCPoint1[16440] = {X 336.4675, Y 19.1512, Z -1.3333, A 0.000, B 0.000, C 0.000 }
gfCNCPoint1[16441] = {X 335.6668, Y 19.6018, Z -1.3333, A 0.000, B 0.000, C 0.000 }
gfCNCPoint1[16442] = {X 334.7878, Y 19.8694, Z -1.3333, A 0.000, B 0.000, C 0.000 }
gfCNCPoint1[16443] = {X 333.8718, Y 19.9414, Z -1.3333, A 0.000, B 0.000, C 0.000 }
gfCNCPoint1[16444] = {X 332.9618, Y 19.8143, Z -1.3333, A 0.000, B 0.000, C 0.000 }
gfCNCPoint1[16445] = {X 332.1006, Y 19.4942, Z -1.3333, A 0.000, B 0.000, C 0.000 }
gfCNCPoint1[16446] = {X 331.3285, Y 18.9960, Z -1.3333, A 0.000, B 0.000, C 0.000 }
gfCNCPoint1[16447] = {X 330.6819, Y 18.3433, Z -1.3333, A 0.000, B 0.000, C 0.000 }
gfCNCPoint1[16448] = {X 330.1911, Y 17.5665, Z -1.3333, A 0.000, B 0.000, C 0.000 }
gfCNCPoint1[16449] = {X 326.6662, Y 10.3152, Z -1.3333, A 0.000, B 0.000, C 0.000 }
gfCNCPoint1[16450] = {X 326.3374, Y 9.3676, Z -1.3333, A 0.000, B 0.000, C 0.000 }
gfCNCPoint1[16451] = {X 326.2405, Y 8.3693, Z -1.3333, A 0.000, B 0.000, C 0.000 }
gfCNCPoint1[16452] = {X 326.3807, Y 7.3762, Z -1.3333, A 0.000, B 0.000, C 0.000 }
gfCNCPoint1[16453] = {X 326.7504, Y 6.4438, Z -1.3333, A 0.000, B 0.000, C 0.000 }
gfCNCPoint1[16454] = {X 327.3287, Y 5.6243, Z -1.3333, A 0.000, B 0.000, C 0.000 }
gfCNCPoint1[16455] = {X 328.0833, Y 4.9636, Z -1.3333, A 0.000, B 0.000, C 0.000 }
gfCNCPoint1[16456] = {X 328.7533, Y 4.5047, Z -1.3333, A 0.000, B 0.000, C 0.000 }
gfCNCPoint1[16457] = {X 329.6263, Y 4.0541, Z -1.3333, A 0.000, B 0.000, C 0.000 }
gfCNCPoint1[16458] = {X 330.5794, Y 3.8165, Z -1.3333, A 0.000, B 0.000, C 0.000 }
gfCNCPoint1[16459] = {X 331.5617, Y 3.8047, Z -1.3333, A 0.000, B 0.000, C 0.000 }
gfCNCPoint1[16460] = {X 332.5203, Y 4.0191, Z -1.3333, A 0.000, B 0.000, C 0.000 }
gfCNCPoint1[16461] = {X 334.0184, Y 3.1813, Z -1.3333, A 0.000, B 0.000, C 0.000 }
gfCNCPoint1[16462] = {X 335.5645, Y 2.4358, Z -1.3333, A 0.000, B 0.000, C 0.000 }
gfCNCPoint1[16463] = {X 337.6942, Y 1.5718, Z -1.3333, A 0.000, B 0.000, C 0.000 }
gfCNCPoint1[16464] = {X 339.8914, Y 0.8978, Z -1.3333, A 0.000, B 0.000, C 0.000 }
gfCNCPoint1[16465] = {X 342.1392, Y 0.4189, Z -1.3333, A 0.000, B 0.000, C 0.000 }
gfCNCPoint1[16466] = {X 344.4203, Y 0.1388, Z -1.3333, A 0.000, B 0.000, C 0.000 }
gfCNCPoint1[16467] = {X 346.7173, Y 0.0598, Z -1.3333, A 0.000, B 0.000, C 0.000 }
gfCNCPoint1[16468] = {X 349.0123, Y 0.1823, Z -1.3333, A 0.000, B 0.000, C 0.000 }
gfCNCPoint1[16469] = {X 351.2877, Y 0.5054, Z -1.3333, A 0.000, B 0.000, C 0.000 }
gfCNCPoint1[16470] = {X 351.5709, Y 0.5577, Z -1.3333, A 0.000, B 0.000, C 0.000 }
gfCNCPoint1[16471] = {X 352.2967, Y -3.3759, Z -1.3333, A 0.000, B 0.000, C 0.000 }
gfCNCPoint1[16472] = {X 351.5563, Y 0.6363, Z -1.3333, A 0.000, B 0.000, C 0.000 }
gfCNCPoint1[16473] = {X 351.8381, Y 0.6883, Z -1.3333, A 0.000, B 0.000, C 0.000 }
gfCNCPoint1[16474] = {X 353.7576, Y 1.1707, Z -1.3333, A 0.000, B 0.000, C 0.000 }
gfCNCPoint1[16475] = {X 355.6228, Y 1.8328, Z -1.3333, A 0.000, B 0.000, C 0.000 }
gfCNCPoint1[16476] = {X 357.4168, Y 2.6686, Z -1.3333, A 0.000, B 0.000, C 0.000 }
gfCNCPoint1[16477] = {X 359.1236, Y 3.6706, Z -1.3333, A 0.000, B 0.000, C 0.000 }
gfCNCPoint1[16478] = {X 360.7279, Y 4.8297, Z -1.3333, A 0.000, B 0.000, C 0.000 }
gfCNCPoint1[16479] = {X 362.2151, Y 6.1357, Z -1.3333, A 0.000, B 0.000, C 0.000 }
gfCNCPoint1[16480] = {X 363.5719, Y 7.5766, Z -1.3333, A 0.000, B 0.000, C 0.000 }
gfCNCPoint1[16481] = {X 365.0323, Y 9.4612, Z -1.3333, A 0.000, B 0.000, C 0.000 }
gfCNCPoint1[16482] = {X 366.3030, Y 11.4785, Z -1.3333, A 0.000, B 0.000, C 0.000 }
gfCNCPoint1[16483] = {X 367.3722, Y 13.6096, Z -1.3333, A 0.000, B 0.000, C 0.000 }
gfCNCPoint1[16484] = {X 368.2297, Y 15.8343, Z -1.3333, A 0.000, B 0.000, C 0.000 }
gfCNCPoint1[16485] = {X 368.8674, Y 18.1316, Z -1.3333, A 0.000, B 0.000, C 0.000 }
gfCNCPoint1[16486] = {X 369.3436, Y 20.7493, Z -1.3333, A 0.000, B 0.000, C 0.000 }
gfCNCPoint1[16487] = {X 369.5971, Y 23.3978, Z -1.3333, A 0.000, B 0.000, C 0.000 }
gfCNCPoint1[16488] = {X 369.6260, Y 26.0584, Z -1.3333, A 0.000, B 0.000, C 0.000 }
gfCNCPoint1[16489] = {X 369.4301, Y 28.7118, Z -1.3333, A 0.000, B 0.000, C 0.000 }
gfCNCPoint1[16490] = {X 369.0109, Y 31.3392, Z -1.3333, A 0.000, B 0.000, C 0.000 }
gfCNCPoint1[16491] = {X 368.4905, Y 33.4302, Z -1.3333, A 0.000, B 0.000, C 0.000 }
gfCNCPoint1[16492] = {X 367.7873, Y 35.4669, Z -1.3333, A 0.000, B 0.000, C 0.000 }
gfCNCPoint1[16493] = {X 366.9068, Y 37.4336, Z -1.3333, A 0.000, B 0.000, C 0.000 }
gfCNCPoint1[16494] = {X 365.8559, Y 39.3147, Z -1.3333, A 0.000, B 0.000, C 0.000 }
gfCNCPoint1[16495] = {X 364.6428, Y 41.0955, Z -1.3333, A 0.000, B 0.000, C 0.000 }
gfCNCPoint1[16496] = {X 363.4249, Y 42.5965, Z -1.3333, A 0.000, B 0.000, C 0.000 }
gfCNCPoint1[16497] = {X 362.0800, Y 43.9849, Z -1.3333, A 0.000, B 0.000, C 0.000 }
gfCNCPoint1[16498] = {X 360.6185, Y 45.2500, Z -1.3333, A 0.000, B 0.000, C 0.000 }
gfCNCPoint1[16499] = {X 359.0517, Y 46.3821, Z -1.3333, A 0.000, B 0.000, C 0.000 }
gfCNCPoint1[16500] = {X 357.3916, Y 47.3724, Z -1.3333, A 0.000, B 0.000, C 0.000 }
gfCNCPoint1[16501] = {X 355.4448, Y 48.2562, Z -1.3333, A 0.000, B 0.000, C 0.000 }
gfCNCPoint1[16502] = {X 353.4227, Y 48.9511, Z -1.3333, A 0.000, B 0.000, C 0.000 }
gfCNCPoint1[16503] = {X 351.3438, Y 49.4507, Z -1.3333, A 0.000, B 0.000, C 0.000 }
gfCNCPoint1[16504] = {X 349.2268, Y 49.7504, Z -1.3333, A 0.000, B 0.000, C 0.000 }
gfCNCPoint1[16505] = {X 347.0909, Y 49.8476, Z -1.3333, A 0.000, B 0.000, C 0.000 }
gfCNCPoint1[16506] = {X 345.0381, Y 49.8132, Z -1.3333, A 0.000, B 0.000, C 0.000 }
gfCNCPoint1[16507] = {X 342.9961, Y 49.6008, Z -1.3333, A 0.000, B 0.000, C 0.000 }
gfCNCPoint1[16508] = {X 340.9801, Y 49.2121, Z -1.3333, A 0.000, B 0.000, C 0.000 }
gfCNCPoint1[16509] = {X 339.0055, Y 48.6500, Z -1.3333, A 0.000, B 0.000, C 0.000 }
gfCNCPoint1[16510] = {X 337.0871, Y 47.9188, Z -1.3333, A 0.000, B 0.000, C 0.000 }
gfCNCPoint1[16511] = {X 335.2393, Y 47.0239, Z -1.3333, A 0.000, B 0.000, C 0.000 }
gfCNCPoint1[16512] = {X 333.6470, Y 46.0382, Z -1.3333, A 0.000, B 0.000, C 0.000 }
gfCNCPoint1[16513] = {X 332.1366, Y 44.9311, Z -1.3333, A 0.000, B 0.000, C 0.000 }
gfCNCPoint1[16514] = {X 330.7174, Y 43.7094, Z -1.3333, A 0.000, B 0.000, C 0.000 }
gfCNCPoint1[16515] = {X 329.7932, Y 43.7230, Z -1.3333, A 0.000, B 0.000, C 0.000 }
gfCNCPoint1[16516] = {X 328.8888, Y 43.5323, Z -1.3333, A 0.000, B 0.000, C 0.000 }
gfCNCPoint1[16517] = {X 328.0488, Y 43.1465, Z -1.3333, A 0.000, B 0.000, C 0.000 }
gfCNCPoint1[16518] = {X 327.3148, Y 42.5847, Z -1.3333, A 0.000, B 0.000, C 0.000 }
gfCNCPoint1[16519] = {X 326.6925, Y 41.9780, Z -1.3333, A 0.000, B 0.000, C 0.000 }
gfCNCPoint1[16520] = {X 326.0873, Y 41.2331, Z -1.3333, A 0.000, B 0.000, C 0.000 }
gfCNCPoint1[16521] = {X 325.6690, Y 40.3693, Z -1.3333, A 0.000, B 0.000, C 0.000 }
gfCNCPoint1[16522] = {X 325.4597, Y 39.4326, Z -1.3333, A 0.000, B 0.000, C 0.000 }
gfCNCPoint1[16523] = {X 325.4707, Y 38.4730, Z -1.3333, A 0.000, B 0.000, C 0.000 }
gfCNCPoint1[16524] = {X 325.7013, Y 37.5413, Z -1.3333, A 0.000, B 0.000, C 0.000 }
gfCNCPoint1[16525] = {X 326.1392, Y 36.6874, Z -1.3333, A 0.000, B 0.000, C 0.000 }
gfCNCPoint1[16526] = {X 330.3969, Y 30.3216, Z -1.3333, A 0.000, B 0.000, C 0.000 }
gfCNCPoint1[16527] = {X 330.9792, Y 29.6411, Z -1.3333, A 0.000, B 0.000, C 0.000 }
gfCNCPoint1[16528] = {X 331.6937, Y 29.1010, Z -1.3333, A 0.000, B 0.000, C 0.000 }
gfCNCPoint1[16529] = {X 332.5073, Y 28.7264, Z -1.3333, A 0.000, B 0.000, C 0.000 }
gfCNCPoint1[16530] = {X 333.3822, Y 28.5346, Z -1.3333, A 0.000, B 0.000, C 0.000 }
gfCNCPoint1[16531] = {X 334.2779, Y 28.5345, Z -1.3333, A 0.000, B 0.000, C 0.000 }
gfCNCPoint1[16532] = {X 335.1528, Y 28.7261, Z -1.3333, A 0.000, B 0.000, C 0.000 }
gfCNCPoint1[16533] = {X 335.9664, Y 29.1006, Z -1.3333, A 0.000, B 0.000, C 0.000 }
gfCNCPoint1[16534] = {X 336.6810, Y 29.6405, Z -1.3333, A 0.000, B 0.000, C 0.000 }
gfCNCPoint1[16535] = {X 337.3163, Y 30.2523, Z -1.3333, A 0.000, B 0.000, C 0.000 }
gfCNCPoint1[16536] = {X 337.8308, Y 30.8659, Z -1.3333, A 0.000, B 0.000, C 0.000 }
gfCNCPoint1[16537] = {X 338.2182, Y 31.5667, Z -1.3333, A 0.000, B 0.000, C 0.000 }
gfCNCPoint1[16538] = {X 338.4642, Y 32.3287, Z -1.3333, A 0.000, B 0.000, C 0.000 }
gfCNCPoint1[16539] = {X 338.5597, Y 33.1237, Z -1.3333, A 0.000, B 0.000, C 0.000 }
gfCNCPoint1[16540] = {X 338.5011, Y 33.9223, Z -1.3333, A 0.000, B 0.000, C 0.000 }
gfCNCPoint1[16541] = {X 339.2990, Y 34.6503, Z -1.3333, A 0.000, B 0.000, C 0.000 }
gfCNCPoint1[16542] = {X 340.1347, Y 35.3347, Z -1.3333, A 0.000, B 0.000, C 0.000 }
gfCNCPoint1[16543] = {X 341.4512, Y 36.1998, Z -1.3333, A 0.000, B 0.000, C 0.000 }
gfCNCPoint1[16544] = {X 342.8798, Y 36.8637, Z -1.3333, A 0.000, B 0.000, C 0.000 }
gfCNCPoint1[16545] = {X 344.3899, Y 37.3121, Z -1.3333, A 0.000, B 0.000, C 0.000 }
gfCNCPoint1[16546] = {X 345.9493, Y 37.5356, Z -1.3333, A 0.000, B 0.000, C 0.000 }
gfCNCPoint1[16547] = {X 347.5246, Y 37.5293, Z -1.3333, A 0.000, B 0.000, C 0.000 }
gfCNCPoint1[16548] = {X 348.7034, Y 37.3906, Z -1.3333, A 0.000, B 0.000, C 0.000 }
gfCNCPoint1[16549] = {X 349.8538, Y 37.0989, Z -1.3333, A 0.000, B 0.000, C 0.000 }
gfCNCPoint1[16550] = {X 350.9563, Y 36.6593, Z -1.3333, A 0.000, B 0.000, C 0.000 }
gfCNCPoint1[16551] = {X 351.9917, Y 36.0794, Z -1.3333, A 0.000, B 0.000, C 0.000 }
gfCNCPoint1[16552] = {X 352.9425, Y 35.3690, Z -1.3333, A 0.000, B 0.000, C 0.000 }
gfCNCPoint1[16553] = {X 354.1081, Y 34.2338, Z -1.3333, A 0.000, B 0.000, C 0.000 }
gfCNCPoint1[16554] = {X 355.1169, Y 32.9574, Z -1.3333, A 0.000, B 0.000, C 0.000 }
gfCNCPoint1[16555] = {X 355.9520, Y 31.5611, Z -1.3333, A 0.000, B 0.000, C 0.000 }
gfCNCPoint1[16556] = {X 356.5993, Y 30.0684, Z -1.3333, A 0.000, B 0.000, C 0.000 }
gfCNCPoint1[16557] = {X 357.0479, Y 28.5045, Z -1.3333, A 0.000, B 0.000, C 0.000 }
gfCNCPoint1[16558] = {X 357.3237, Y 26.8012, Z -1.3333, A 0.000, B 0.000, C 0.000 }
gfCNCPoint1[16559] = {X 357.4360, Y 25.0793, Z -1.3333, A 0.000, B 0.000, C 0.000 }
gfCNCPoint1[16560] = {X 357.3839, Y 23.3545, Z -1.3333, A 0.000, B 0.000, C 0.000 }
gfCNCPoint1[16561] = {X 357.1678, Y 21.6425, Z -1.3333, A 0.000, B 0.000, C 0.000 }
gfCNCPoint1[16562] = {X 356.8270, Y 20.1740, Z -1.3333, A 0.000, B 0.000, C 0.000 }
gfCNCPoint1[16563] = {X 356.3071, Y 18.7589, Z -1.3333, A 0.000, B 0.000, C 0.000 }
gfCNCPoint1[16564] = {X 355.6161, Y 17.4190, Z -1.3333, A 0.000, B 0.000, C 0.000 }
gfCNCPoint1[16565] = {X 354.7647, Y 16.1748, Z -1.3333, A 0.000, B 0.000, C 0.000 }
gfCNCPoint1[16566] = {X 353.8634, Y 15.1696, Z -1.3333, A 0.000, B 0.000, C 0.000 }
gfCNCPoint1[16567] = {X 352.8273, Y 14.3038, Z -1.3333, A 0.000, B 0.000, C 0.000 }
gfCNCPoint1[16568] = {X 351.6779, Y 13.5955, Z -1.3333, A 0.000, B 0.000, C 0.000 }
gfCNCPoint1[16569] = {X 350.4390, Y 13.0590, Z -1.3333, A 0.000, B 0.000, C 0.000 }
gfCNCPoint1[16570] = {X 349.1359, Y 12.7056, Z -1.3333, A 0.000, B 0.000, C 0.000 }
gfCNCPoint1[16571] = {X 347.5974, Y 12.5003, Z -1.3333, A 0.000, B 0.000, C 0.000 }
gfCNCPoint1[16572] = {X 346.0456, Y 12.4723, Z -1.3333, A 0.000, B 0.000, C 0.000 }
gfCNCPoint1[16573] = {X 344.5007, Y 12.6221, Z -1.3333, A 0.000, B 0.000, C 0.000 }
gfCNCPoint1[16574] = {X 342.9831, Y 12.9476, Z -1.3333, A 0.000, B 0.000, C 0.000 }
gfCNCPoint1[16575] = {X 341.5127, Y 13.4446, Z -1.3333, A 0.000, B 0.000, C 0.000 }
gfCNCPoint1[16576] = {X 340.1088, Y 14.1066, Z -1.3333, A 0.000, B 0.000, C 0.000 }
gfCNCPoint1[16577] = {X 338.7899, Y 14.9248, Z -1.3333, A 0.000, B 0.000, C 0.000 }
gfCNCPoint1[16578] = {X 338.7950, Y 14.9999, Z -1.3333, A 0.000, B 0.000, C 0.000 }
gfCNCPoint1[16579] = {X 338.7601, Y 15.8161, Z -1.3333, A 0.000, B 0.000, C 0.000 }
gfCNCPoint1[16580] = {X 338.5663, Y 16.6097, Z -1.3333, A 0.000, B 0.000, C 0.000 }
gfCNCPoint1[16581] = {X 338.2211, Y 17.3501, Z -1.3333, A 0.000, B 0.000, C 0.000 }
gfCNCPoint1[16582] = {X 337.7379, Y 18.0088, Z -1.3333, A 0.000, B 0.000, C 0.000 }
gfCNCPoint1[16583] = {X 337.1353, Y 18.5603, Z -1.3333, A 0.000, B 0.000, C 0.000 }
gfCNCPoint1[16584] = {X 336.4209, Y 19.0861, Z -1.3333, A 0.000, B 0.000, C 0.000 }
gfCNCPoint1[16585] = {X 335.6353, Y 19.5283, Z -1.3333, A 0.000, B 0.000, C 0.000 }
gfCNCPoint1[16586] = {X 334.7729, Y 19.7908, Z -1.3333, A 0.000, B 0.000, C 0.000 }
gfCNCPoint1[16587] = {X 333.8742, Y 19.8614, Z -1.3333, A 0.000, B 0.000, C 0.000 }
gfCNCPoint1[16588] = {X 332.9814, Y 19.7367, Z -1.3333, A 0.000, B 0.000, C 0.000 }
gfCNCPoint1[16589] = {X 332.1364, Y 19.4226, Z -1.3333, A 0.000, B 0.000, C 0.000 }
gfCNCPoint1[16590] = {X 331.3789, Y 18.9339, Z -1.3333, A 0.000, B 0.000, C 0.000 }
gfCNCPoint1[16591] = {X 330.7445, Y 18.2934, Z -1.3333, A 0.000, B 0.000, C 0.000 }
gfCNCPoint1[16592] = {X 330.2630, Y 17.5314, Z -1.3333, A 0.000, B 0.000, C 0.000 }
gfCNCPoint1[16593] = {X 326.7381, Y 10.2803, Z -1.3333, A 0.000, B 0.000, C 0.000 }
gfCNCPoint1[16594] = {X 326.4156, Y 9.3505, Z -1.3333, A 0.000, B 0.000, C 0.000 }
gfCNCPoint1[16595] = {X 326.3205, Y 8.3711, Z -1.3333, A 0.000, B 0.000, C 0.000 }
gfCNCPoint1[16596] = {X 326.4581, Y 7.3967, Z -1.3333, A 0.000, B 0.000, C 0.000 }
gfCNCPoint1[16597] = {X 326.8207, Y 6.4819, Z -1.3333, A 0.000, B 0.000, C 0.000 }
gfCNCPoint1[16598] = {X 327.3881, Y 5.6778, Z -1.3333, A 0.000, B 0.000, C 0.000 }
gfCNCPoint1[16599] = {X 328.1285, Y 5.0296, Z -1.3333, A 0.000, B 0.000, C 0.000 }
gfCNCPoint1[16600] = {X 328.7983, Y 4.5709, Z -1.3333, A 0.000, B 0.000, C 0.000 }
gfCNCPoint1[16601] = {X 329.6634, Y 4.1256, Z -1.3333, A 0.000, B 0.000, C 0.000 }
gfCNCPoint1[16602] = {X 330.6083, Y 3.8935, Z -1.3333, A 0.000, B 0.000, C 0.000 }
gfCNCPoint1[16603] = {X 331.5813, Y 3.8872, Z -1.3333, A 0.000, B 0.000, C 0.000 }
gfCNCPoint1[16604] = {X 332.5292, Y 4.1071, Z -1.3333, A 0.000, B 0.000, C 0.000 }
gfCNCPoint1[16605] = {X 334.0388, Y 3.2608, Z -1.3333, A 0.000, B 0.000, C 0.000 }
gfCNCPoint1[16606] = {X 335.5974, Y 2.5087, Z -1.3333, A 0.000, B 0.000, C 0.000 }
gfCNCPoint1[16607] = {X 337.7207, Y 1.6473, Z -1.3333, A 0.000, B 0.000, C 0.000 }
gfCNCPoint1[16608] = {X 339.9112, Y 0.9753, Z -1.3333, A 0.000, B 0.000, C 0.000 }
gfCNCPoint1[16609] = {X 342.1523, Y 0.4978, Z -1.3333, A 0.000, B 0.000, C 0.000 }
gfCNCPoint1[16610] = {X 344.4265, Y 0.2186, Z -1.3333, A 0.000, B 0.000, C 0.000 }
gfCNCPoint1[16611] = {X 346.7165, Y 0.1398, Z -1.3333, A 0.000, B 0.000, C 0.000 }
gfCNCPoint1[16612] = {X 349.0046, Y 0.2619, Z -1.3333, A 0.000, B 0.000, C 0.000 }
gfCNCPoint1[16613] = {X 351.2731, Y 0.5841, Z -1.3333, A 0.000, B 0.000, C 0.000 }
gfCNCPoint1[16614] = {X 351.5563, Y 0.6363, Z -1.3333, A 0.000, B 0.000, C 0.000 }
gfCNCPoint1[16615] = {X 352.2822, Y -3.2973, Z -1.3333, A 0.000, B 0.000, C 0.000 }
gfCNCPoint1[16616] = {X 351.5418, Y 0.7150, Z -1.3333, A 0.000, B 0.000, C 0.000 }
gfCNCPoint1[16617] = {X 351.8229, Y 0.7669, Z -1.3333, A 0.000, B 0.000, C 0.000 }
gfCNCPoint1[16618] = {X 353.7350, Y 1.2475, Z -1.3333, A 0.000, B 0.000, C 0.000 }
gfCNCPoint1[16619] = {X 355.5929, Y 1.9070, Z -1.3333, A 0.000, B 0.000, C 0.000 }
gfCNCPoint1[16620] = {X 357.3800, Y 2.7396, Z -1.3333, A 0.000, B 0.000, C 0.000 }
gfCNCPoint1[16621] = {X 359.0802, Y 3.7377, Z -1.3333, A 0.000, B 0.000, C 0.000 }
gfCNCPoint1[16622] = {X 360.6782, Y 4.8924, Z -1.3333, A 0.000, B 0.000, C 0.000 }
gfCNCPoint1[16623] = {X 362.1596, Y 6.1933, Z -1.3333, A 0.000, B 0.000, C 0.000 }
gfCNCPoint1[16624] = {X 363.5111, Y 7.6286, Z -1.3333, A 0.000, B 0.000, C 0.000 }
gfCNCPoint1[16625] = {X 364.9667, Y 9.5071, Z -1.3333, A 0.000, B 0.000, C 0.000 }
gfCNCPoint1[16626] = {X 366.2333, Y 11.5179, Z -1.3333, A 0.000, B 0.000, C 0.000 }
gfCNCPoint1[16627] = {X 367.2990, Y 13.6420, Z -1.3333, A 0.000, B 0.000, C 0.000 }
gfCNCPoint1[16628] = {X 368.1537, Y 15.8594, Z -1.3333, A 0.000, B 0.000, C 0.000 }
gfCNCPoint1[16629] = {X 368.7894, Y 18.1492, Z -1.3333, A 0.000, B 0.000, C 0.000 }
gfCNCPoint1[16630] = {X 369.2644, Y 20.7603, Z -1.3333, A 0.000, B 0.000, C 0.000 }
gfCNCPoint1[16631] = {X 369.5172, Y 23.4021, Z -1.3333, A 0.000, B 0.000, C 0.000 }
gfCNCPoint1[16632] = {X 369.5460, Y 26.0559, Z -1.3333, A 0.000, B 0.000, C 0.000 }
gfCNCPoint1[16633] = {X 369.3507, Y 28.7026, Z -1.3333, A 0.000, B 0.000, C 0.000 }
gfCNCPoint1[16634] = {X 368.9325, Y 31.3233, Z -1.3333, A 0.000, B 0.000, C 0.000 }
gfCNCPoint1[16635] = {X 368.4138, Y 33.4074, Z -1.3333, A 0.000, B 0.000, C 0.000 }
gfCNCPoint1[16636] = {X 367.7129, Y 35.4375, Z -1.3333, A 0.000, B 0.000, C 0.000 }
gfCNCPoint1[16637] = {X 366.8353, Y 37.3977, Z -1.3333, A 0.000, B 0.000, C 0.000 }
gfCNCPoint1[16638] = {X 365.7878, Y 39.2727, Z -1.3333, A 0.000, B 0.000, C 0.000 }
gfCNCPoint1[16639] = {X 364.5787, Y 41.0477, Z -1.3333, A 0.000, B 0.000, C 0.000 }
gfCNCPoint1[16640] = {X 363.3653, Y 42.5432, Z -1.3333, A 0.000, B 0.000, C 0.000 }
gfCNCPoint1[16641] = {X 362.0254, Y 43.9265, Z -1.3333, A 0.000, B 0.000, C 0.000 }
gfCNCPoint1[16642] = {X 360.5693, Y 45.1869, Z -1.3333, A 0.000, B 0.000, C 0.000 }
gfCNCPoint1[16643] = {X 359.0083, Y 46.3149, Z -1.3333, A 0.000, B 0.000, C 0.000 }
gfCNCPoint1[16644] = {X 357.3544, Y 47.3015, Z -1.3333, A 0.000, B 0.000, C 0.000 }
gfCNCPoint1[16645] = {X 355.4144, Y 48.1822, Z -1.3333, A 0.000, B 0.000, C 0.000 }
gfCNCPoint1[16646] = {X 353.3994, Y 48.8745, Z -1.3333, A 0.000, B 0.000, C 0.000 }
gfCNCPoint1[16647] = {X 351.3278, Y 49.3723, Z -1.3333, A 0.000, B 0.000, C 0.000 }
gfCNCPoint1[16648] = {X 349.2183, Y 49.6708, Z -1.3333, A 0.000, B 0.000, C 0.000 }
gfCNCPoint1[16649] = {X 347.0899, Y 49.7676, Z -1.3333, A 0.000, B 0.000, C 0.000 }
gfCNCPoint1[16650] = {X 345.0440, Y 49.7334, Z -1.3333, A 0.000, B 0.000, C 0.000 }
gfCNCPoint1[16651] = {X 343.0088, Y 49.5218, Z -1.3333, A 0.000, B 0.000, C 0.000 }
gfCNCPoint1[16652] = {X 340.9996, Y 49.1345, Z -1.3333, A 0.000, B 0.000, C 0.000 }
gfCNCPoint1[16653] = {X 339.0316, Y 48.5744, Z -1.3333, A 0.000, B 0.000, C 0.000 }
gfCNCPoint1[16654] = {X 337.1196, Y 47.8457, Z -1.3333, A 0.000, B 0.000, C 0.000 }
gfCNCPoint1[16655] = {X 335.2780, Y 46.9539, Z -1.3333, A 0.000, B 0.000, C 0.000 }
gfCNCPoint1[16656] = {X 333.6809, Y 45.9646, Z -1.3333, A 0.000, B 0.000, C 0.000 }
gfCNCPoint1[16657] = {X 332.1666, Y 44.8527, Z -1.3333, A 0.000, B 0.000, C 0.000 }
gfCNCPoint1[16658] = {X 330.7444, Y 43.6252, Z -1.3333, A 0.000, B 0.000, C 0.000 }
gfCNCPoint1[16659] = {X 329.8288, Y 43.6460, Z -1.3333, A 0.000, B 0.000, C 0.000 }
gfCNCPoint1[16660] = {X 328.9316, Y 43.4621, Z -1.3333, A 0.000, B 0.000, C 0.000 }
gfCNCPoint1[16661] = {X 328.0981, Y 43.0827, Z -1.3333, A 0.000, B 0.000, C 0.000 }
gfCNCPoint1[16662] = {X 327.3701, Y 42.5270, Z -1.3333, A 0.000, B 0.000, C 0.000 }
gfCNCPoint1[16663] = {X 326.7483, Y 41.9207, Z -1.3333, A 0.000, B 0.000, C 0.000 }
gfCNCPoint1[16664] = {X 326.1548, Y 41.1901, Z -1.3333, A 0.000, B 0.000, C 0.000 }
gfCNCPoint1[16665] = {X 325.7445, Y 40.3430, Z -1.3333, A 0.000, B 0.000, C 0.000 }
gfCNCPoint1[16666] = {X 325.5393, Y 39.4243, Z -1.3333, A 0.000, B 0.000, C 0.000 }
gfCNCPoint1[16667] = {X 325.5500, Y 38.4831, Z -1.3333, A 0.000, B 0.000, C 0.000 }
gfCNCPoint1[16668] = {X 325.7762, Y 37.5694, Z -1.3333, A 0.000, B 0.000, C 0.000 }
gfCNCPoint1[16669] = {X 326.2057, Y 36.7318, Z -1.3333, A 0.000, B 0.000, C 0.000 }
gfCNCPoint1[16670] = {X 330.4629, Y 30.3668, Z -1.3333, A 0.000, B 0.000, C 0.000 }
gfCNCPoint1[16671] = {X 331.0340, Y 29.6994, Z -1.3333, A 0.000, B 0.000, C 0.000 }
gfCNCPoint1[16672] = {X 331.7347, Y 29.1697, Z -1.3333, A 0.000, B 0.000, C 0.000 }
gfCNCPoint1[16673] = {X 332.5326, Y 28.8023, Z -1.3333, A 0.000, B 0.000, C 0.000 }
gfCNCPoint1[16674] = {X 333.3906, Y 28.6141, Z -1.3333, A 0.000, B 0.000, C 0.000 }
gfCNCPoint1[16675] = {X 334.2690, Y 28.6140, Z -1.3333, A 0.000, B 0.000, C 0.000 }
gfCNCPoint1[16676] = {X 335.1270, Y 28.8018, Z -1.3333, A 0.000, B 0.000, C 0.000 }
gfCNCPoint1[16677] = {X 335.9250, Y 29.1690, Z -1.3333, A 0.000, B 0.000, C 0.000 }
gfCNCPoint1[16678] = {X 336.6259, Y 29.6985, Z -1.3333, A 0.000, B 0.000, C 0.000 }
gfCNCPoint1[16679] = {X 337.2602, Y 30.3094, Z -1.3333, A 0.000, B 0.000, C 0.000 }
gfCNCPoint1[16680] = {X 337.7696, Y 30.9181, Z -1.3333, A 0.000, B 0.000, C 0.000 }
gfCNCPoint1[16681] = {X 338.1515, Y 31.6139, Z -1.3333, A 0.000, B 0.000, C 0.000 }
gfCNCPoint1[16682] = {X 338.3914, Y 32.3705, Z -1.3333, A 0.000, B 0.000, C 0.000 }
gfCNCPoint1[16683] = {X 338.4804, Y 33.1593, Z -1.3333, A 0.000, B 0.000, C 0.000 }
gfCNCPoint1[16684] = {X 338.4149, Y 33.9503, Z -1.3333, A 0.000, B 0.000, C 0.000 }
gfCNCPoint1[16685] = {X 339.2306, Y 34.6969, Z -1.3333, A 0.000, B 0.000, C 0.000 }
gfCNCPoint1[16686] = {X 340.0858, Y 35.3980, Z -1.3333, A 0.000, B 0.000, C 0.000 }
gfCNCPoint1[16687] = {X 341.4119, Y 36.2695, Z -1.3333, A 0.000, B 0.000, C 0.000 }
gfCNCPoint1[16688] = {X 342.8510, Y 36.9383, Z -1.3333, A 0.000, B 0.000, C 0.000 }
gfCNCPoint1[16689] = {X 344.3721, Y 37.3901, Z -1.3333, A 0.000, B 0.000, C 0.000 }
gfCNCPoint1[16690] = {X 345.9429, Y 37.6154, Z -1.3333, A 0.000, B 0.000, C 0.000 }
gfCNCPoint1[16691] = {X 347.5298, Y 37.6092, Z -1.3333, A 0.000, B 0.000, C 0.000 }
gfCNCPoint1[16692] = {X 348.7187, Y 37.4691, Z -1.3333, A 0.000, B 0.000, C 0.000 }
gfCNCPoint1[16693] = {X 349.8791, Y 37.1748, Z -1.3333, A 0.000, B 0.000, C 0.000 }
gfCNCPoint1[16694] = {X 350.9911, Y 36.7314, Z -1.3333, A 0.000, B 0.000, C 0.000 }
gfCNCPoint1[16695] = {X 352.0355, Y 36.1463, Z -1.3333, A 0.000, B 0.000, C 0.000 }
gfCNCPoint1[16696] = {X 352.9945, Y 35.4298, Z -1.3333, A 0.000, B 0.000, C 0.000 }
gfCNCPoint1[16697] = {X 354.1675, Y 34.2874, Z -1.3333, A 0.000, B 0.000, C 0.000 }
gfCNCPoint1[16698] = {X 355.1828, Y 33.0027, Z -1.3333, A 0.000, B 0.000, C 0.000 }
gfCNCPoint1[16699] = {X 356.0232, Y 31.5975, Z -1.3333, A 0.000, B 0.000, C 0.000 }
gfCNCPoint1[16700] = {X 356.6747, Y 30.0953, Z -1.3333, A 0.000, B 0.000, C 0.000 }
gfCNCPoint1[16701] = {X 357.1262, Y 28.5213, Z -1.3333, A 0.000, B 0.000, C 0.000 }
gfCNCPoint1[16702] = {X 357.4032, Y 26.8104, Z -1.3333, A 0.000, B 0.000, C 0.000 }
gfCNCPoint1[16703] = {X 357.5160, Y 25.0808, Z -1.3333, A 0.000, B 0.000, C 0.000 }
gfCNCPoint1[16704] = {X 357.4637, Y 23.3484, Z -1.3333, A 0.000, B 0.000, C 0.000 }
gfCNCPoint1[16705] = {X 357.2466, Y 21.6288, Z -1.3333, A 0.000, B 0.000, C 0.000 }
gfCNCPoint1[16706] = {X 356.9035, Y 20.1507, Z -1.3333, A 0.000, B 0.000, C 0.000 }
gfCNCPoint1[16707] = {X 356.3802, Y 18.7264, Z -1.3333, A 0.000, B 0.000, C 0.000 }
gfCNCPoint1[16708] = {X 355.6847, Y 17.3778, Z -1.3333, A 0.000, B 0.000, C 0.000 }
gfCNCPoint1[16709] = {X 354.8278, Y 16.1256, Z -1.3333, A 0.000, B 0.000, C 0.000 }
gfCNCPoint1[16710] = {X 353.9188, Y 15.1119, Z -1.3333, A 0.000, B 0.000, C 0.000 }
gfCNCPoint1[16711] = {X 352.8739, Y 14.2388, Z -1.3333, A 0.000, B 0.000, C 0.000 }
gfCNCPoint1[16712] = {X 351.7148, Y 13.5244, Z -1.3333, A 0.000, B 0.000, C 0.000 }
gfCNCPoint1[16713] = {X 350.4653, Y 12.9835, Z -1.3333, A 0.000, B 0.000, C 0.000 }
gfCNCPoint1[16714] = {X 349.1511, Y 12.6271, Z -1.3333, A 0.000, B 0.000, C 0.000 }
gfCNCPoint1[16715] = {X 347.5971, Y 12.4200, Z -1.3333, A 0.000, B 0.000, C 0.000 }
gfCNCPoint1[16716] = {X 346.0296, Y 12.3929, Z -1.3333, A 0.000, B 0.000, C 0.000 }
gfCNCPoint1[16717] = {X 344.4694, Y 12.5460, Z -1.3333, A 0.000, B 0.000, C 0.000 }
gfCNCPoint1[16718] = {X 342.9371, Y 12.8773, Z -1.3333, A 0.000, B 0.000, C 0.000 }
gfCNCPoint1[16719] = {X 341.4529, Y 13.3825, Z -1.3333, A 0.000, B 0.000, C 0.000 }
gfCNCPoint1[16720] = {X 340.0367, Y 14.0548, Z -1.3333, A 0.000, B 0.000, C 0.000 }
gfCNCPoint1[16721] = {X 338.7070, Y 14.8854, Z -1.3333, A 0.000, B 0.000, C 0.000 }
gfCNCPoint1[16722] = {X 338.7152, Y 15.0048, Z -1.3333, A 0.000, B 0.000, C 0.000 }
gfCNCPoint1[16723] = {X 338.6808, Y 15.8052, Z -1.3333, A 0.000, B 0.000, C 0.000 }
gfCNCPoint1[16724] = {X 338.4907, Y 16.5834, Z -1.3333, A 0.000, B 0.000, C 0.000 }
gfCNCPoint1[16725] = {X 338.1522, Y 17.3095, Z -1.3333, A 0.000, B 0.000, C 0.000 }
gfCNCPoint1[16726] = {X 337.6783, Y 17.9554, Z -1.3333, A 0.000, B 0.000, C 0.000 }
gfCNCPoint1[16727] = {X 337.0874, Y 18.4963, Z -1.3333, A 0.000, B 0.000, C 0.000 }
gfCNCPoint1[16728] = {X 336.3744, Y 19.0211, Z -1.3333, A 0.000, B 0.000, C 0.000 }
gfCNCPoint1[16729] = {X 335.6039, Y 19.4547, Z -1.3333, A 0.000, B 0.000, C 0.000 }
gfCNCPoint1[16730] = {X 334.7580, Y 19.7122, Z -1.3333, A 0.000, B 0.000, C 0.000 }
gfCNCPoint1[16731] = {X 333.8766, Y 19.7814, Z -1.3333, A 0.000, B 0.000, C 0.000 }
gfCNCPoint1[16732] = {X 333.0010, Y 19.6592, Z -1.3333, A 0.000, B 0.000, C 0.000 }
gfCNCPoint1[16733] = {X 332.1722, Y 19.3511, Z -1.3333, A 0.000, B 0.000, C 0.000 }
gfCNCPoint1[16734] = {X 331.4293, Y 18.8718, Z -1.3333, A 0.000, B 0.000, C 0.000 }
gfCNCPoint1[16735] = {X 330.8071, Y 18.2436, Z -1.3333, A 0.000, B 0.000, C 0.000 }
gfCNCPoint1[16736] = {X 330.3348, Y 17.4962, Z -1.3333, A 0.000, B 0.000, C 0.000 }
gfCNCPoint1[16737] = {X 326.8101, Y 10.2453, Z -1.3333, A 0.000, B 0.000, C 0.000 }
gfCNCPoint1[16738] = {X 326.4937, Y 9.3334, Z -1.3333, A 0.000, B 0.000, C 0.000 }
gfCNCPoint1[16739] = {X 326.4004, Y 8.3728, Z -1.3333, A 0.000, B 0.000, C 0.000 }
gfCNCPoint1[16740] = {X 326.5354, Y 7.4171, Z -1.3333, A 0.000, B 0.000, C 0.000 }
gfCNCPoint1[16741] = {X 326.8911, Y 6.5199, Z -1.3333, A 0.000, B 0.000, C 0.000 }
gfCNCPoint1[16742] = {X 327.4476, Y 5.7314, Z -1.3333, A 0.000, B 0.000, C 0.000 }
gfCNCPoint1[16743] = {X 328.1737, Y 5.0956, Z -1.3333, A 0.000, B 0.000, C 0.000 }
gfCNCPoint1[16744] = {X 328.8432, Y 4.6371, Z -1.3333, A 0.000, B 0.000, C 0.000 }
gfCNCPoint1[16745] = {X 329.7006, Y 4.1972, Z -1.3333, A 0.000, B 0.000, C 0.000 }
gfCNCPoint1[16746] = {X 330.6372, Y 3.9706, Z -1.3333, A 0.000, B 0.000, C 0.000 }
gfCNCPoint1[16747] = {X 331.6008, Y 3.9700, Z -1.3333, A 0.000, B 0.000, C 0.000 }
gfCNCPoint1[16748] = {X 332.5377, Y 4.1954, Z -1.3333, A 0.000, B 0.000, C 0.000 }
gfCNCPoint1[16749] = {X 334.0590, Y 3.3405, Z -1.3333, A 0.000, B 0.000, C 0.000 }
gfCNCPoint1[16750] = {X 335.6304, Y 2.5816, Z -1.3333, A 0.000, B 0.000, C 0.000 }
gfCNCPoint1[16751] = {X 337.7472, Y 1.7228, Z -1.3333, A 0.000, B 0.000, C 0.000 }
gfCNCPoint1[16752] = {X 339.9311, Y 1.0528, Z -1.3333, A 0.000, B 0.000, C 0.000 }
gfCNCPoint1[16753] = {X 342.1653, Y 0.5768, Z -1.3333, A 0.000, B 0.000, C 0.000 }
gfCNCPoint1[16754] = {X 344.4327, Y 0.2984, Z -1.3333, A 0.000, B 0.000, C 0.000 }
gfCNCPoint1[16755] = {X 346.7157, Y 0.2198, Z -1.3333, A 0.000, B 0.000, C 0.000 }
gfCNCPoint1[16756] = {X 348.9968, Y 0.3415, Z -1.3333, A 0.000, B 0.000, C 0.000 }
gfCNCPoint1[16757] = {X 351.2585, Y 0.6627, Z -1.3333, A 0.000, B 0.000, C 0.000 }
gfCNCPoint1[16758] = {X 351.5418, Y 0.7150, Z -1.3333, A 0.000, B 0.000, C 0.000 }
gfCNCPoint1[16759] = {X 352.2677, Y -3.2186, Z -1.3333, A 0.000, B 0.000, C 0.000 }
gfCNCPoint1[16760] = {X 351.5273, Y 0.7937, Z -1.3333, A 0.000, B 0.000, C 0.000 }
gfCNCPoint1[16761] = {X 351.8078, Y 0.8454, Z -1.3333, A 0.000, B 0.000, C 0.000 }
gfCNCPoint1[16762] = {X 353.7123, Y 1.3242, Z -1.3333, A 0.000, B 0.000, C 0.000 }
gfCNCPoint1[16763] = {X 355.5630, Y 1.9812, Z -1.3333, A 0.000, B 0.000, C 0.000 }
gfCNCPoint1[16764] = {X 357.3431, Y 2.8106, Z -1.3333, A 0.000, B 0.000, C 0.000 }
gfCNCPoint1[16765] = {X 359.0367, Y 3.8049, Z -1.3333, A 0.000, B 0.000, C 0.000 }
gfCNCPoint1[16766] = {X 360.6284, Y 4.9551, Z -1.3333, A 0.000, B 0.000, C 0.000 }
gfCNCPoint1[16767] = {X 362.1041, Y 6.2509, Z -1.3333, A 0.000, B 0.000, C 0.000 }
gfCNCPoint1[16768] = {X 363.4503, Y 7.6806, Z -1.3333, A 0.000, B 0.000, C 0.000 }
gfCNCPoint1[16769] = {X 364.9012, Y 9.5530, Z -1.3333, A 0.000, B 0.000, C 0.000 }
gfCNCPoint1[16770] = {X 366.1637, Y 11.5572, Z -1.3333, A 0.000, B 0.000, C 0.000 }
gfCNCPoint1[16771] = {X 367.2258, Y 13.6743, Z -1.3333, A 0.000, B 0.000, C 0.000 }
gfCNCPoint1[16772] = {X 368.0777, Y 15.8845, Z -1.3333, A 0.000, B 0.000, C 0.000 }
gfCNCPoint1[16773] = {X 368.7113, Y 18.1668, Z -1.3333, A 0.000, B 0.000, C 0.000 }
gfCNCPoint1[16774] = {X 369.1851, Y 20.7713, Z -1.3333, A 0.000, B 0.000, C 0.000 }
gfCNCPoint1[16775] = {X 369.4373, Y 23.4064, Z -1.3333, A 0.000, B 0.000, C 0.000 }
gfCNCPoint1[16776] = {X 369.4661, Y 26.0534, Z -1.3333, A 0.000, B 0.000, C 0.000 }
gfCNCPoint1[16777] = {X 369.2712, Y 28.6933, Z -1.3333, A 0.000, B 0.000, C 0.000 }
gfCNCPoint1[16778] = {X 368.8541, Y 31.3074, Z -1.3333, A 0.000, B 0.000, C 0.000 }
gfCNCPoint1[16779] = {X 368.3371, Y 33.3847, Z -1.3333, A 0.000, B 0.000, C 0.000 }
gfCNCPoint1[16780] = {X 367.6385, Y 35.4081, Z -1.3333, A 0.000, B 0.000, C 0.000 }
gfCNCPoint1[16781] = {X 366.7637, Y 37.3619, Z -1.3333, A 0.000, B 0.000, C 0.000 }
gfCNCPoint1[16782] = {X 365.7197, Y 39.2307, Z -1.3333, A 0.000, B 0.000, C 0.000 }
gfCNCPoint1[16783] = {X 364.5146, Y 40.9999, Z -1.3333, A 0.000, B 0.000, C 0.000 }
gfCNCPoint1[16784] = {X 363.3056, Y 42.4898, Z -1.3333, A 0.000, B 0.000, C 0.000 }
gfCNCPoint1[16785] = {X 361.9707, Y 43.8680, Z -1.3333, A 0.000, B 0.000, C 0.000 }
gfCNCPoint1[16786] = {X 360.5201, Y 45.1239, Z -1.3333, A 0.000, B 0.000, C 0.000 }
gfCNCPoint1[16787] = {X 358.9649, Y 46.2476, Z -1.3333, A 0.000, B 0.000, C 0.000 }
gfCNCPoint1[16788] = {X 357.3172, Y 47.2307, Z -1.3333, A 0.000, B 0.000, C 0.000 }
gfCNCPoint1[16789] = {X 355.3840, Y 48.1082, Z -1.3333, A 0.000, B 0.000, C 0.000 }
gfCNCPoint1[16790] = {X 353.3762, Y 48.7980, Z -1.3333, A 0.000, B 0.000, C 0.000 }
gfCNCPoint1[16791] = {X 351.3118, Y 49.2939, Z -1.3333, A 0.000, B 0.000, C 0.000 }
gfCNCPoint1[16792] = {X 349.2098, Y 49.5913, Z -1.3333, A 0.000, B 0.000, C 0.000 }
gfCNCPoint1[16793] = {X 347.0889, Y 49.6876, Z -1.3333, A 0.000, B 0.000, C 0.000 }
gfCNCPoint1[16794] = {X 345.0499, Y 49.6536, Z -1.3333, A 0.000, B 0.000, C 0.000 }
gfCNCPoint1[16795] = {X 343.0216, Y 49.4428, Z -1.3333, A 0.000, B 0.000, C 0.000 }
gfCNCPoint1[16796] = {X 341.0191, Y 49.0569, Z -1.3333, A 0.000, B 0.000, C 0.000 }
gfCNCPoint1[16797] = {X 339.0577, Y 48.4988, Z -1.3333, A 0.000, B 0.000, C 0.000 }
gfCNCPoint1[16798] = {X 337.1521, Y 47.7726, Z -1.3333, A 0.000, B 0.000, C 0.000 }
gfCNCPoint1[16799] = {X 335.3167, Y 46.8838, Z -1.3333, A 0.000, B 0.000, C 0.000 }
gfCNCPoint1[16800] = {X 333.7147, Y 45.8908, Z -1.3333, A 0.000, B 0.000, C 0.000 }
gfCNCPoint1[16801] = {X 332.1963, Y 44.7741, Z -1.3333, A 0.000, B 0.000, C 0.000 }
gfCNCPoint1[16802] = {X 330.7711, Y 43.5406, Z -1.3333, A 0.000, B 0.000, C 0.000 }
gfCNCPoint1[16803] = {X 329.8559, Y 43.5681, Z -1.3333, A 0.000, B 0.000, C 0.000 }
gfCNCPoint1[16804] = {X 328.9583, Y 43.3867, Z -1.3333, A 0.000, B 0.000, C 0.000 }
gfCNCPoint1[16805] = {X 328.1256, Y 43.0059, Z -1.3333, A 0.000, B 0.000, C 0.000 }
gfCNCPoint1[16806] = {X 327.4012, Y 42.4458, Z -1.3333, A 0.000, B 0.000, C 0.000 }
gfCNCPoint1[16807] = {X 326.8042, Y 41.8634, Z -1.3333, A 0.000, B 0.000, C 0.000 }
gfCNCPoint1[16808] = {X 326.2223, Y 41.1472, Z -1.3333, A 0.000, B 0.000, C 0.000 }
gfCNCPoint1[16809] = {X 325.8201, Y 40.3166, Z -1.3333, A 0.000, B 0.000, C 0.000 }
gfCNCPoint1[16810] = {X 325.6189, Y 39.4160, Z -1.3333, A 0.000, B 0.000, C 0.000 }
gfCNCPoint1[16811] = {X 325.6294, Y 38.4932, Z -1.3333, A 0.000, B 0.000, C 0.000 }
gfCNCPoint1[16812] = {X 325.8511, Y 37.5974, Z -1.3333, A 0.000, B 0.000, C 0.000 }
gfCNCPoint1[16813] = {X 326.2722, Y 36.7763, Z -1.3333, A 0.000, B 0.000, C 0.000 }
gfCNCPoint1[16814] = {X 330.5290, Y 30.4119, Z -1.3333, A 0.000, B 0.000, C 0.000 }
gfCNCPoint1[16815] = {X 331.0932, Y 29.7535, Z -1.3333, A 0.000, B 0.000, C 0.000 }
gfCNCPoint1[16816] = {X 331.7861, Y 29.2322, Z -1.3333, A 0.000, B 0.000, C 0.000 }
gfCNCPoint1[16817] = {X 332.5750, Y 28.8724, Z -1.3333, A 0.000, B 0.000, C 0.000 }
gfCNCPoint1[16818] = {X 333.4230, Y 28.6911, Z -1.3333, A 0.000, B 0.000, C 0.000 }
gfCNCPoint1[16819] = {X 334.2901, Y 28.6968, Z -1.3333, A 0.000, B 0.000, C 0.000 }
gfCNCPoint1[16820] = {X 335.1355, Y 28.8892, Z -1.3333, A 0.000, B 0.000, C 0.000 }
gfCNCPoint1[16821] = {X 335.9197, Y 29.2593, Z -1.3333, A 0.000, B 0.000, C 0.000 }
gfCNCPoint1[16822] = {X 336.6057, Y 29.7897, Z -1.3333, A 0.000, B 0.000, C 0.000 }
gfCNCPoint1[16823] = {X 337.2041, Y 30.3665, Z -1.3333, A 0.000, B 0.000, C 0.000 }
gfCNCPoint1[16824] = {X 337.7083, Y 30.9703, Z -1.3333, A 0.000, B 0.000, C 0.000 }
gfCNCPoint1[16825] = {X 338.0846, Y 31.6611, Z -1.3333, A 0.000, B 0.000, C 0.000 }
gfCNCPoint1[16826] = {X 338.3184, Y 32.4122, Z -1.3333, A 0.000, B 0.000, C 0.000 }
gfCNCPoint1[16827] = {X 338.4007, Y 33.1945, Z -1.3333, A 0.000, B 0.000, C 0.000 }
gfCNCPoint1[16828] = {X 338.3283, Y 33.9779, Z -1.3333, A 0.000, B 0.000, C 0.000 }
gfCNCPoint1[16829] = {X 339.1620, Y 34.7433, Z -1.3333, A 0.000, B 0.000, C 0.000 }
gfCNCPoint1[16830] = {X 340.0369, Y 35.4613, Z -1.3333, A 0.000, B 0.000, C 0.000 }
gfCNCPoint1[16831] = {X 341.2949, Y 36.2949, Z -1.3333, A 0.000, B 0.000, C 0.000 }
gfCNCPoint1[16832] = {X 342.6557, Y 36.9473, Z -1.3333, A 0.000, B 0.000, C 0.000 }
gfCNCPoint1[16833] = {X 344.0934, Y 37.4062, Z -1.3333, A 0.000, B 0.000, C 0.000 }
gfCNCPoint1[16834] = {X 345.5806, Y 37.6627, Z -1.3333, A 0.000, B 0.000, C 0.000 }
gfCNCPoint1[16835] = {X 347.0889, Y 37.7121, Z -1.3333, A 0.000, B 0.000, C 0.000 }
gfCNCPoint1[16836] = {X 347.5339, Y 37.6891, Z -1.3333, A 0.000, B 0.000, C 0.000 }
gfCNCPoint1[16837] = {X 348.7332, Y 37.5478, Z -1.3333, A 0.000, B 0.000, C 0.000 }
gfCNCPoint1[16838] = {X 349.9038, Y 37.2509, Z -1.3333, A 0.000, B 0.000, C 0.000 }
gfCNCPoint1[16839] = {X 351.0255, Y 36.8036, Z -1.3333, A 0.000, B 0.000, C 0.000 }
gfCNCPoint1[16840] = {X 352.0791, Y 36.2134, Z -1.3333, A 0.000, B 0.000, C 0.000 }
